    IF (Direction = ComDirection.ROB_TO_PLC)
    THEN  
      // calculate sequence payload length
      CalculateSequencePayloadMax := ( _parCfg.Com.TelegramLengthRobToPlc - _cyclicDataLength );
    END_IF
    

  SequenceFlag.SECONDARY_SEQUENCE :
  
    IF (Direction = ComDirection.PLC_TO_ROB)
    THEN  
      // calculate sequence payload length
      CalculateSequencePayloadMax := (( _parCfg.Com.TelegramLengthPlcToRob - _cyclicDataLength ) / 2);
    END_IF

    IF (Direction = ComDirection.ROB_TO_PLC)
    THEN  
      // calculate sequence payload length
      CalculateSequencePayloadMax := (( _parCfg.Com.TelegramLengthRobToPlc - _cyclicDataLength ) / 2);
    END_IF

    
END_CASE
                
END_METHOD

METHOD CalculateSequencePayloadStartAdr : UINT
VAR_IN_OUT
  /// Robot assignment of function
  AxesGroup : AxesGroup;
END_VAR
VAR_INPUT
  /// Communication direction
  Direction : ComDirection;
  /// Sequeunce
  Sequence : SequenceFlag;  
END_VAR

VAR
  /// Length of the cyclic header
 _cyclicDataLength      : UINT;
  /// Length of the sequnce payload
 _sequencePayloadLength : UINT;
END_VAR
                  // calculate cyclic header length
_cyclicDataLength := CalculateCyclicDataLength(AxesGroup := AxesGroup, Direction := Direction);

CASE (Sequence) 
OF

  SequenceFlag.PRIMARY_SEQUENCE   : 
  
    // return start address
    CalculateSequencePayloadStartAdr := _cyclicDataLength;

  SequenceFlag.SECONDARY_SEQUENCE :
  
    // calculate sequence payload max
   _sequencePayloadLength 
     := CalculateSequencePayloadMax( AxesGroup := AxesGroup, 
                                     Direction := Direction, 
                                     Sequence  := Sequence );
                                     
    // return start address
    CalculateSequencePayloadStartAdr := _cyclicDataLength + _sequencePayloadLength;
    
END_CASE
                
END_METHOD

METHOD PRIVATE CalculateTelegramLengthPlcToRob : UINT
VAR_IN_OUT
  /// Robot assignment of function
  AxesGroup : AxesGroup;
END_VAR
VAR
  /// length of the cyclic data block
 _cyclicDataLength : UINT;
END_VAR
                  _cyclicDataLength := CalculateCyclicDataLength(AxesGroup := AxesGroup, Direction := ComDirection.PLC_TO_ROB); 


IF ( _parCfg.Com.TwoSequences )
THEN
  CalculateTelegramLengthPlcToRob := _cyclicDataLength
                                    + SIZEOF(Telegram.PlcToRob.Sequence[  PRIMARY_SEQUENCE].Header)
                                    +       (Telegram.PlcToRob.Sequence[  PRIMARY_SEQUENCE].Header.PayloadLength)
                                    + SIZEOF(Telegram.PlcToRob.Sequence[SECONDARY_SEQUENCE].Header)
                                    +       (Telegram.PlcToRob.Sequence[SECONDARY_SEQUENCE].Header.PayloadLength)
                                    + SIZEOF(Telegram.PlcToRob.Footer);  
ELSE
  CalculateTelegramLengthPlcToRob := _cyclicDataLength
                                    + SIZEOF(Telegram.PlcToRob.Sequence[PRIMARY_SEQUENCE].Header)
                                    +       (Telegram.PlcToRob.Sequence[PRIMARY_SEQUENCE].Header.PayloadLength)
                                    + SIZEOF(Telegram.PlcToRob.Footer);
END_IF
                
END_METHOD

METHOD PROTECTED CheckParameterChanged : BOOL
VAR_IN_OUT
  /// Robot assignment of function
  AxesGroup    : AxesGroup; 
END_VAR

VAR
  /// internal index for loops
 _idx : DINT;
END_VAR
                  // Check initialization is already done ?
IF ( NOT Initialized )
THEN
  CheckParameterChanged := FALSE;
  RETURN;
END_IF

// compare memory 
CheckParameterChanged := ( SysDepMemCmp(pData1 := ADR(ParCfg), pData2 := ADR(_parCfg), DataLen := SIZEOF(ParCfg)) <> RobotLibraryConstants.OK );

FOR _idx := SyncTime.DURING_START_UP TO SyncTime.AFTER_START_UP
DO
  // Check Tool SyncMode changed ? 
  IF ( _parCfg.Plc.Parameter.SynchronizationModes.Tool[_idx] <> ParCfg.Plc.Parameter.SynchronizationModes.Tool[_idx] )
  THEN
    // Set info
    SetInfo( InfoID := RobotLibraryInfoIdEnum.INFO_CHANGE_TOOL_SYNC_MODE_TO_NEGATIVE_ONLY_AT_PLC_START_ALLOWED, Overwrite := TRUE);
     
    // Create log entry
    CreateLogMessagePara3( Timestamp   := SystemTime,
                           MessageType := MessageType.CMD,
                           Severity    := Severity.INFO,
                           MessageCode := 0,
                           MessageText := 'SyncMode.Tool[{1}] changed from {2} to {3}, but this is only allowed at PLC start',
                           Para1       := SYNC_TIME_TO_STRING(_idx),
                           Para2       := SYNC_MODE_TO_STRING( ParCfg.Plc.Parameter.SynchronizationModes.Tool[_idx]),
                           Para3       := SYNC_MODE_TO_STRING(_parCfg.Plc.Parameter.SynchronizationModes.Tool[_idx]));   
  END_IF
  
  
  // Check Frame SyncMode changed ? 
  IF ( _parCfg.Plc.Parameter.SynchronizationModes.Frame[_idx] <> ParCfg.Plc.Parameter.SynchronizationModes.Frame[_idx] )
  THEN
    // Set info
    SetInfo( InfoID := RobotLibraryInfoIdEnum.INFO_CHANGE_FRAME_SYNC_MODE_TO_NEGATIVE_ONLY_AT_PLC_START_ALLOWED, Overwrite :=  TRUE);
     
    // Create log entry
    CreateLogMessagePara3( Timestamp   := SystemTime,
                           MessageType := MessageType.CMD,
                           Severity    := Severity.INFO,
                           MessageCode := 0,
                           MessageText := 'SyncMode.Frame[{1}] changed from {2} to {3}, but this is only allowed at PLC start',
                           Para1       := SYNC_TIME_TO_STRING(_idx),
                           Para2       := SYNC_MODE_TO_STRING( ParCfg.Plc.Parameter.SynchronizationModes.Frame[_idx]),
                           Para3       := SYNC_MODE_TO_STRING(_parCfg.Plc.Parameter.SynchronizationModes.Frame[_idx]));   
  END_IF
  
  
  // Check Load SyncMode changed ? 
  IF ( _parCfg.Plc.Parameter.SynchronizationModes.Load[_idx] <> ParCfg.Plc.Parameter.SynchronizationModes.Load[_idx] )
  THEN
    // Set info
    SetInfo( InfoID := RobotLibraryInfoIdEnum.INFO_CHANGE_LOAD_SYNC_MODE_TO_NEGATIVE_ONLY_AT_PLC_START_ALLOWED, Overwrite := TRUE);
     
    // Create log entry
    CreateLogMessagePara3( Timestamp   := SystemTime,
                           MessageType := MessageType.CMD,
                           Severity    := Severity.INFO,
                           MessageCode := 0,
                           MessageText := 'SyncMode.Load[{1}] changed from {2} to {3}, but this is only allowed at PLC start',
                           Para1       := SYNC_TIME_TO_STRING(_idx),
                           Para2       := SYNC_MODE_TO_STRING( ParCfg.Plc.Parameter.SynchronizationModes.Load[_idx]),
                           Para3       := SYNC_MODE_TO_STRING(_parCfg.Plc.Parameter.SynchronizationModes.Load[_idx]));   
  END_IF
  
  
  // Check WorkAreas SyncMode changed ? 
  IF ( _parCfg.Plc.Parameter.SynchronizationModes.WorkAreas[_idx] <> ParCfg.Plc.Parameter.SynchronizationModes.WorkAreas[_idx] )
  THEN
    // Set info
    SetInfo( InfoID := RobotLibraryInfoIdEnum.INFO_CHANGE_WORK_AREA_SYNC_MODE_TO_NEGATIVE_ONLY_AT_PLC_START_ALLOWED, Overwrite := TRUE);
     
    // Create log entry
    CreateLogMessagePara3( Timestamp   := SystemTime,
                           MessageType := MessageType.CMD,
                           Severity    := Severity.INFO,
                           MessageCode := 0,
                           MessageText := 'SyncMode.WorkAreas[{1}] changed from {2} to {3}, but this is only allowed at PLC start',
                           Para1       := SYNC_TIME_TO_STRING(_idx),
                           Para2       := SYNC_MODE_TO_STRING( ParCfg.Plc.Parameter.SynchronizationModes.WorkAreas[_idx]),
                           Para3       := SYNC_MODE_TO_STRING(_parCfg.Plc.Parameter.SynchronizationModes.WorkAreas[_idx]));   
  END_IF

  // Check SWLimits SyncMode changed ? 
  IF ( _parCfg.Plc.Parameter.SynchronizationModes.SWLimits[_idx] <> ParCfg.Plc.Parameter.SynchronizationModes.SWLimits[_idx] )
  THEN
    // Set info
    SetInfo( InfoID := RobotLibraryInfoIdEnum.INFO_CHANGE_SWLIMITS_SYNC_MODE_TO_NEGATIVE_ONLY_AT_PLC_START_ALLOWED, Overwrite := TRUE);
     
    // Create log entry
    CreateLogMessagePara3( Timestamp   := SystemTime,
                           MessageType := MessageType.CMD,
                           Severity    := Severity.INFO,
                           MessageCode := 0,
                           MessageText := 'SyncMode.SWLimits[{1}] changed from {2} to {3}, but this is only allowed at PLC start',
                           Para1       := SYNC_TIME_TO_STRING(_idx),
                           Para2       := SYNC_MODE_TO_STRING( ParCfg.Plc.Parameter.SynchronizationModes.SWLimits[_idx]),
                           Para3       := SYNC_MODE_TO_STRING(_parCfg.Plc.Parameter.SynchronizationModes.SWLimits[_idx]));   
  END_IF
  
 
  // Check DefaultDynamics SyncMode changed ? 
  IF ( _parCfg.Plc.Parameter.SynchronizationModes.DefaultDynamics[_idx] <> ParCfg.Plc.Parameter.SynchronizationModes.DefaultDynamics[_idx] )
  THEN
    // Set info
    SetInfo( InfoID := RobotLibraryInfoIdEnum.INFO_CHANGE_DEFAULT_DYNAMICS_SYNC_MODE_TO_NEGATIVE_ONLY_AT_PLC_START_ALLOWED, Overwrite := TRUE);
     
    // Create log entry
    CreateLogMessagePara3( Timestamp   := SystemTime,
                           MessageType := MessageType.CMD,
                           Severity    := Severity.INFO,
                           MessageCode := 0,
                           MessageText := 'SyncMode.DefaultDynamics[{1}] changed from {2} to {3}, but this is only allowed at PLC start',
                           Para1       := SYNC_TIME_TO_STRING(_idx),
                           Para2       := SYNC_MODE_TO_STRING( ParCfg.Plc.Parameter.SynchronizationModes.DefaultDynamics[_idx]),
                           Para3       := SYNC_MODE_TO_STRING(_parCfg.Plc.Parameter.SynchronizationModes.DefaultDynamics[_idx]));   
  END_IF
  
  
  // Check ReferenceDynamics SyncMode changed ?
  IF ( _parCfg.Plc.Parameter.SynchronizationModes.ReferenceDynamics[_idx] <> ParCfg.Plc.Parameter.SynchronizationModes.ReferenceDynamics[_idx] )
  THEN
    // Set info
    SetInfo(InfoID := RobotLibraryInfoIdEnum.INFO_CHANGE_REFERENCE_DYNAMICS_SYNC_MODE_TO_NEGATIVE_ONLY_AT_PLC_START_ALLOWED, Overwrite := TRUE );
     
    // Create log entry
    CreateLogMessagePara3( Timestamp   := SystemTime,
                           MessageType := MessageType.CMD,
                           Severity    := Severity.INFO,
                           MessageCode := 0,
                           MessageText := 'SyncMode.ReferenceDynamics[{1}] changed from {2} to {3}, but this is only allowed at PLC start',
                           Para1       := SYNC_TIME_TO_STRING(_idx),
                           Para2       := SYNC_MODE_TO_STRING( ParCfg.Plc.Parameter.SynchronizationModes.ReferenceDynamics[_idx]),
                           Para3       := SYNC_MODE_TO_STRING(_parCfg.Plc.Parameter.SynchronizationModes.ReferenceDynamics[_idx]));   
  END_IF

END_FOR


// Check Plc.OptionalCyclic changed ? 
IF ( PlcOptionalCyclicToUint(_parCfg.Plc.OptionalCyclic) <> PlcOptionalCyclicToUint(ParCfg.Plc.OptionalCyclic ))
THEN
  // Set error
  SetError( ErrorID := RobotLibraryErrorIdEnum.ERR_TELEGRAM_NUMBER_CHANGED_AFTER_INIT, Overwrite := TRUE );
   
  // Create log entry
  CreateLogMessagePara2( Timestamp   := SystemTime,
                         MessageType := MessageType.CMD,
                         Severity    := Severity.ERROR,
                         MessageCode := 0,
                         MessageText := 'ParCfg.Plc.OptionalCyclic changed after initialization from {1} to {2} -> Reinitialize by disabling and enabling the RobotTask',
                         Para1       := WORD_TO_STRING_BIN(PlcOptionalCyclicToUint(_parCfg.Plc.OptionalCyclic)),
                         Para2       := WORD_TO_STRING_BIN(PlcOptionalCyclicToUint( ParCfg.Plc.OptionalCyclic)));   
END_IF


// Check Rob.OptionalCyclic changed ? 
IF ( RobOptionalCyclicToUint(_parCfg.Rob.OptionalCyclic) <> RobOptionalCyclicToUint(ParCfg.Rob.OptionalCyclic ))
THEN
  // Set error
  SetError( ErrorID := RobotLibraryErrorIdEnum.ERR_TELEGRAM_NUMBER_CHANGED_AFTER_INIT, Overwrite := TRUE );
   
  // Create log entry
  CreateLogMessagePara2( Timestamp   := SystemTime,
                         MessageType := MessageType.CMD,
                         Severity    := Severity.ERROR,
                         MessageCode := 0,
                         MessageText := 'ParCfg.Rob.OptionalCyclic changed after initialization from {1} to {2} -> Reinitialize by disabling and enabling the RobotTask',
                         Para1       := WORD_TO_STRING_BIN(RobOptionalCyclicToUint(_parCfg.Rob.OptionalCyclic)),
                         Para2       := WORD_TO_STRING_BIN(RobOptionalCyclicToUint( ParCfg.Rob.OptionalCyclic)));   
END_IF

                
END_METHOD

METHOD PROTECTED CheckParameterValid : BOOL
VAR_IN_OUT
  /// Robot assignment of function
  AxesGroup : AxesGroup; 
END_VAR
                  // init return value
CheckParameterValid := TRUE;


// Check ParCfg.Com.TelegramLengthPlcToRob
IF ( ParCfg.Com.TelegramLengthPlcToRob < 128 )
THEN
  // Set Warning
  SetWarning( WarningID := RobotLibraryWarningIdEnum.WARN_ACYCLIC_RANGE_PLC_TO_ROB_VERY_SMALL, Overwrite := TRUE );
END_IF

// Check ParCfg.Com.TelegramLengthRobToPlc
IF ( ParCfg.Com.TelegramLengthRobToPlc < 128 )
THEN
  // Set Warning
  SetWarning( WarningID := RobotLibraryWarningIdEnum.WARN_ACYCLIC_RANGE_ROB_TO_PLC_VERY_SMALL, Overwrite := TRUE );
END_IF



// Region ParCfg.Com {{{

// Check LifeSignTimeout
IF ( ParCfg.Com.LifeSignTimeOut < T#10MS )
THEN
  // set to valid min value
  ParCfg.Com.LifeSignTimeOut := T#10MS;
 
  // Set info
  SetInfo( InfoID := RobotLibraryInfoIdEnum.INFO_LIFESIGN_TIMEOUT_TO_SMALL_AND_SET_TO_10MS, Overwrite := TRUE);
   
  // Create log entry
  CreateLogMessagePara1 ( Timestamp   := SystemTime,
                          MessageType := MessageType.CMD,
                          Severity    := Severity.INFO,
                          MessageCode := 0,
                          MessageText := 'LifeSignTimeout to small and set from {1}ms to 10ms',
                          Para1       := TIME_TO_STRING(ParCfg.Com.LifeSignTimeOut));                          
END_IF


// Check ParCfg.Com.TelegramLengthPlcToRob
IF (( ParCfg.Com.TelegramLengthPlcToRob < 64                  ) OR
    ( ParCfg.Com.TelegramLengthPlcToRob > ROBOT_OUT_DATA_SIZE ))
THEN
  // parameter(s) not valid
  CheckParameterValid := FALSE;

  // Set error
  SetError( ErrorID := RobotLibraryErrorIdEnum.ERR_TELEGRAM_LENGTH_MISMATCH_0x80A3, Overwrite := TRUE );
   
  // Create log entry
  CreateLogMessagePara1 ( Timestamp   := SystemTime,
                          MessageType := MessageType.CMD,
                          Severity    := Severity.INFO,
                          MessageCode := 0,
                          MessageText :=               'ParCfg.Com.TelegramLengthPlcToRob {1} invalid',
                          Para1       := UINT_TO_STRING(ParCfg.Com.TelegramLengthPlcToRob));
  // no further validation                          
  RETURN;                          
END_IF

// Check ParCfg.Com.TelegramLengthRobToPlc
IF (( ParCfg.Com.TelegramLengthRobToPlc < 64                 ) OR
    ( ParCfg.Com.TelegramLengthRobToPlc > ROBOT_IN_DATA_SIZE ))
THEN
  // parameter(s) not valid
  CheckParameterValid := FALSE;

  // Set error
  SetError( ErrorID := RobotLibraryErrorIdEnum.ERR_TELEGRAM_LENGTH_MISMATCH_0x80A3, Overwrite := TRUE );
   
  // Create log entry
  CreateLogMessagePara1 ( Timestamp   := SystemTime,
                          MessageType := MessageType.CMD,
                          Severity    := Severity.INFO,
                          MessageCode := 0,
                          MessageText :=               'ParCfg.Com.TelegramLengthRobToPlc {1} invalid',
                          Para1       := UINT_TO_STRING(ParCfg.Com.TelegramLengthRobToPlc));
  // no further validation                          
  RETURN;                          
END_IF
// EndRegion }}}

// Region ParCfg.Rob.OptionalCyclic {{{

// Check configuration if optional cyclic CartesianPosition valid ?
IF ( ParCfg.Rob.OptionalCyclic.UseCartesianPosition AND ParCfg.Rob.OptionalCyclic.UseCartesianPositionExt )
THEN
  // set to valid configuration
  ParCfg.Rob.OptionalCyclic.UseCartesianPosition    := TRUE;
  ParCfg.Rob.OptionalCyclic.UseCartesianPositionExt := FALSE;
 
  // Set info
  SetInfo( InfoID := RobotLibraryInfoIdEnum.INFO_RECV_EXT_CART_POS_NOT_USABLE_WITH_RECV_CART_POS, Overwrite := TRUE);
   
  // Create log entry
  CreateLogMessage( Timestamp   := SystemTime,
                    MessageType := MessageType.CMD,
                    Severity    := Severity.INFO,
                    MessageCode := 0,
                    MessageText := 'UseCartesianPosition and UseCartesianPositionExt cannot be configured together -> UseCartesianPosition is automatically activated');
END_IF


// Check configuration if optional cyclic JointPosition valid ?
IF ( ParCfg.Rob.OptionalCyclic.UseJointPosition AND ParCfg.Rob.OptionalCyclic.UseJointPositionExt ) AND FALSE  {warning 'ToDo: Yaskawa need this combination for debugging via JointPosExt '}
THEN
  // set to valid configuration
  ParCfg.Rob.OptionalCyclic.UseJointPosition    := TRUE;
  ParCfg.Rob.OptionalCyclic.UseJointPositionExt := FALSE;
 
  // Set info
  SetInfo( InfoID := RobotLibraryInfoIdEnum.INFO_RECV_EXT_JOINT_POS_NOT_USABLE_WITH_RECV_JOINT_POS, Overwrite := TRUE);
   
  // Create log entry
  CreateLogMessage( Timestamp   := SystemTime,
                    MessageType := MessageType.CMD,
                    Severity    := Severity.INFO,
                    MessageCode := 0,
                    MessageText := 'UseJointPosition and UseJointPositionExt cannot be configured together -> UseJointPosition is automatically activated');
END_IF
// EndRegion }}}

// Region ParCfg.Parameter.SynchronizationModes {{{

// Check ToolData synchronisation mode during startup
IF (( ParCfg.Plc.Parameter.SynchronizationModes.Tool[SyncTime.DURING_START_UP] <  SyncMode.NO_SYNCHRONIZATION ) OR
    ( ParCfg.Plc.Parameter.SynchronizationModes.Tool[SyncTime.DURING_START_UP] >= SyncMode.AUTOMATIC          )) // Automatic is not allowed during startup
THEN
  // parameter(s) not valid
  CheckParameterValid := FALSE;
 
  // Set error
  SetError  ( ErrorID   := RobotLibraryErrorIdEnum.ERR_SYNC_MODE_INVALID             , Overwrite := TRUE ); // own defined error - not in specification
  // Set warning
  SetWarning( WarningID := RobotLibraryWarningIdEnum.WARN_TOOL_DATA_SYNC_MODE_INVALID, Overwrite := TRUE );
   
  // Create log entry
  CreateLogMessagePara1 ( Timestamp   := SystemTime,
                          MessageType := MessageType.CMD,
                          Severity    := Severity.INFO,
                          MessageCode := 0,
                          MessageText :=                    'ParCfg.Plc.Parameter.SynchronizationModes.Tool[SyncTime.DURING_START_UP] invalid SyncMode {1}',
                          Para1       := SYNC_MODE_TO_STRING(ParCfg.Plc.Parameter.SynchronizationModes.Tool[SyncTime.DURING_START_UP]));
  // no further validation                          
  RETURN;                                                    
END_IF

// Check ToolData synchronisation mode after startup
IF (( ParCfg.Plc.Parameter.SynchronizationModes.Tool[SyncTime.AFTER_START_UP] < SyncMode.NO_SYNCHRONIZATION ) OR
    ( ParCfg.Plc.Parameter.SynchronizationModes.Tool[SyncTime.AFTER_START_UP] > SyncMode.AUTOMATIC          ))
THEN
  // parameter(s) not valid
  CheckParameterValid := FALSE;
 
  // Set error
  SetError  ( ErrorID   := RobotLibraryErrorIdEnum.ERR_SYNC_MODE_INVALID             , Overwrite := TRUE); // own defined error - not in specification
  // Set warning
  SetWarning( WarningID := RobotLibraryWarningIdEnum.WARN_TOOL_DATA_SYNC_MODE_INVALID, Overwrite := TRUE);
   
  // Create log entry
  CreateLogMessagePara1 ( Timestamp   := SystemTime,
                          MessageType := MessageType.CMD,
                          Severity    := Severity.INFO,
                          MessageCode := 0,
                          MessageText :=                    'ParCfg.Plc.Parameter.SynchronizationModes.Tool[SyncTime.AFTER_START_UP] invalid SyncMode {1}',
                          Para1       := SYNC_MODE_TO_STRING(ParCfg.Plc.Parameter.SynchronizationModes.Tool[SyncTime.AFTER_START_UP]));
  // no further validation                          
  RETURN;                                                    
END_IF


// Check FrameData synchronisation mode during startup
IF (( ParCfg.Plc.Parameter.SynchronizationModes.Frame[SyncTime.DURING_START_UP] <  SyncMode.NO_SYNCHRONIZATION ) OR
    ( ParCfg.Plc.Parameter.SynchronizationModes.Frame[SyncTime.DURING_START_UP] >= SyncMode.AUTOMATIC          )) // Automatic is not allowed during startup
THEN
  // parameter(s) not valid
  CheckParameterValid := FALSE;
 
  // Set error
  SetError  ( ErrorID   := RobotLibraryErrorIdEnum.ERR_SYNC_MODE_INVALID              , Overwrite := TRUE);// own defined error - not in specification
  // Set warning
  SetWarning( WarningID := RobotLibraryWarningIdEnum.WARN_FRAME_DATA_SYNC_MODE_INVALID, Overwrite := FALSE);
   
  // Create log entry
  CreateLogMessagePara1 ( Timestamp   := SystemTime,
                          MessageType := MessageType.CMD,
                          Severity    := Severity.INFO,
                          MessageCode := 0,
                          MessageText :=                    'ParCfg.Plc.Parameter.SynchronizationModes.Frame[SyncTime.DURING_START_UP] invalid SyncMode {1}',
                          Para1       := SYNC_MODE_TO_STRING(ParCfg.Plc.Parameter.SynchronizationModes.Frame[SyncTime.DURING_START_UP]));
  // no further validation                          
  RETURN;                                                   
END_IF


// Check FrameData synchronisation mode after startup
IF (( ParCfg.Plc.Parameter.SynchronizationModes.Frame[SyncTime.AFTER_START_UP] < SyncMode.NO_SYNCHRONIZATION ) OR
    ( ParCfg.Plc.Parameter.SynchronizationModes.Frame[SyncTime.AFTER_START_UP] > SyncMode.AUTOMATIC          ))
THEN
  // parameter(s) not valid
  CheckParameterValid := FALSE;
 
  // Set error
  SetError  ( ErrorID   := RobotLibraryErrorIdEnum.ERR_SYNC_MODE_INVALID              , Overwrite := TRUE);// own defined error - not in specification
  // Set warning
  SetWarning( WarningID := RobotLibraryWarningIdEnum.WARN_FRAME_DATA_SYNC_MODE_INVALID, Overwrite := TRUE);
   
  // Create log entry
  CreateLogMessagePara1 ( Timestamp   := SystemTime,
                          MessageType := MessageType.CMD,
                          Severity    := Severity.INFO,
                          MessageCode := 0,
                          MessageText :=                    'ParCfg.Plc.Parameter.SynchronizationModes.Frame[SyncTime.AFTER_START_UP] invalid SyncMode {1}',
                          Para1       := SYNC_MODE_TO_STRING(ParCfg.Plc.Parameter.SynchronizationModes.Frame[SyncTime.AFTER_START_UP]));
  // no further validation                          
  RETURN;                                                    
END_IF


// Check LoadData synchronisation mode during startup
IF (( ParCfg.Plc.Parameter.SynchronizationModes.Load[SyncTime.DURING_START_UP] <  SyncMode.NO_SYNCHRONIZATION ) OR
    ( ParCfg.Plc.Parameter.SynchronizationModes.Load[SyncTime.DURING_START_UP] >= SyncMode.AUTOMATIC          )) // Automatic is not allowed during startup
THEN
  // parameter(s) not valid
  CheckParameterValid := FALSE;
 
  // Set error
  SetError   ( ErrorID   := RobotLibraryErrorIdEnum.ERR_SYNC_MODE_INVALID             , Overwrite := TRUE);// own defined error - not in specification
  // Set warning
  SetWarning ( WarningID := RobotLibraryWarningIdEnum.WARN_LOAD_DATA_SYNC_MODE_INVALID, Overwrite := TRUE);
   
  // Create log entry
  CreateLogMessagePara1 ( Timestamp   := SystemTime,
                          MessageType := MessageType.CMD,
                          Severity    := Severity.INFO,
                          MessageCode := 0,
                          MessageText :=                    'ParCfg.Plc.Parameter.SynchronizationModes.Load[SyncTime.DURING_START_UP] invalid SyncMode {1}',
                          Para1       := SYNC_MODE_TO_STRING(ParCfg.Plc.Parameter.SynchronizationModes.Load[SyncTime.DURING_START_UP]));
  // no further validation                          
  RETURN;                          
END_IF


// Check LoadData synchronisation mode after startup
IF (( ParCfg.Plc.Parameter.SynchronizationModes.Load[SyncTime.AFTER_START_UP] < SyncMode.NO_SYNCHRONIZATION ) OR
    ( ParCfg.Plc.Parameter.SynchronizationModes.Load[SyncTime.AFTER_START_UP] > SyncMode.AUTOMATIC          ))
THEN
  // parameter(s) not valid
  CheckParameterValid := FALSE;
 
  // Set error
  SetError  ( ErrorID   := RobotLibraryErrorIdEnum.ERR_SYNC_MODE_INVALID,              Overwrite := TRUE);// own defined error - not in specification
  // Set warning
  SetWarning( WarningID := RobotLibraryWarningIdEnum.WARN_LOAD_DATA_SYNC_MODE_INVALID, Overwrite := TRUE);
   
  // Create log entry
  CreateLogMessagePara1 ( Timestamp   := SystemTime,
                          MessageType := MessageType.CMD,
                          Severity    := Severity.INFO,
                          MessageCode := 0,
                          MessageText :=                    'ParCfg.Plc.Parameter.SynchronizationModes.Load[SyncTime.AFTER_START_UP] invalid SyncMode {1}',
                          Para1       := SYNC_MODE_TO_STRING(ParCfg.Plc.Parameter.SynchronizationModes.Load[SyncTime.AFTER_START_UP]));
  // no further validation                          
  RETURN;                          
END_IF


// Check WorkAreas synchronisation mode during startup
IF (( ParCfg.Plc.Parameter.SynchronizationModes.WorkAreas[SyncTime.DURING_START_UP] <  SyncMode.NO_SYNCHRONIZATION ) OR
    ( ParCfg.Plc.Parameter.SynchronizationModes.WorkAreas[SyncTime.DURING_START_UP] >= SyncMode.AUTOMATIC          )) // Automatic is not allowed during startup
THEN
  // parameter(s) not valid
  CheckParameterValid := FALSE;
 
  // Set error
  SetError  ( ErrorID   := RobotLibraryErrorIdEnum.ERR_SYNC_MODE_INVALID,              Overwrite := TRUE);// own defined error - not in specification
  // Set warning
  SetWarning( WarningID := RobotLibraryWarningIdEnum.WARN_WORK_AREA_SYNC_MODE_INVALID, Overwrite := TRUE);
   
  // Create log entry
  CreateLogMessagePara1 ( Timestamp   := SystemTime,
                          MessageType := MessageType.CMD,
                          Severity    := Severity.INFO,
                          MessageCode := 0,
                          MessageText :=                    'ParCfg.Plc.Parameter.SynchronizationModes.WorkAreas[SyncTime.DURING_START_UP] invalid SyncMode {1}',
                          Para1       := SYNC_MODE_TO_STRING(ParCfg.Plc.Parameter.SynchronizationModes.WorkAreas[SyncTime.DURING_START_UP]));
  // no further validation                          
  RETURN;                          
END_IF


// Check WorkAreas synchronisation mode after startup
IF (( ParCfg.Plc.Parameter.SynchronizationModes.WorkAreas[SyncTime.AFTER_START_UP] < SyncMode.NO_SYNCHRONIZATION ) OR
    ( ParCfg.Plc.Parameter.SynchronizationModes.WorkAreas[SyncTime.AFTER_START_UP] > SyncMode.AUTOMATIC          ))
THEN
  // parameter(s) not valid
  CheckParameterValid := FALSE;
 
  // Set error
  SetError  ( ErrorID   := RobotLibraryErrorIdEnum.ERR_SYNC_MODE_INVALID,              Overwrite := TRUE);// own defined error - not in specification
  // Set warning
  SetWarning( WarningID := RobotLibraryWarningIdEnum.WARN_WORK_AREA_SYNC_MODE_INVALID, Overwrite := TRUE);
   
  // Create log entry
  CreateLogMessagePara1 ( Timestamp   := SystemTime,
                          MessageType := MessageType.CMD,
                          Severity    := Severity.INFO,
                          MessageCode := 0,
                          MessageText :=                    'ParCfg.Plc.Parameter.SynchronizationModes.WorkAreas[SyncTime.AFTER_START_UP] invalid SyncMode {1}',
                          Para1       := SYNC_MODE_TO_STRING(ParCfg.Plc.Parameter.SynchronizationModes.WorkAreas[SyncTime.AFTER_START_UP]));
  // no further validation                          
  RETURN;                          
END_IF


// Check SWLimits synchronisation mode during startup
IF (( ParCfg.Plc.Parameter.SynchronizationModes.SWLimits[SyncTime.DURING_START_UP] <  SyncMode.NO_SYNCHRONIZATION ) OR
    ( ParCfg.Plc.Parameter.SynchronizationModes.SWLimits[SyncTime.DURING_START_UP] >= SyncMode.AUTOMATIC          )) // Automatic is not allowed during startup
THEN
  // parameter(s) not valid
  CheckParameterValid := FALSE;
 
  // Set error
  SetError  ( ErrorID   := RobotLibraryErrorIdEnum.ERR_SYNC_MODE_INVALID,              Overwrite := TRUE);// own defined error - not in specification
  // Set warning
  SetWarning( WarningID := RobotLibraryWarningIdEnum.WARN_SW_LIMITS_SYNC_MODE_INVALID, Overwrite := TRUE);
   
  // Create log entry
  CreateLogMessagePara1 ( Timestamp   := SystemTime,
                          MessageType := MessageType.CMD,
                          Severity    := Severity.INFO,
                          MessageCode := 0,
                          MessageText :=                    'ParCfg.Plc.Parameter.SynchronizationModes.SWLimits[SyncTime.DURING_START_UP] invalid SyncMode {1}',
                          Para1       := SYNC_MODE_TO_STRING(ParCfg.Plc.Parameter.SynchronizationModes.SWLimits[SyncTime.DURING_START_UP]));
  // no further validation                          
  RETURN;                          
END_IF


// Check SWLimits synchronisation mode after startup
IF (( ParCfg.Plc.Parameter.SynchronizationModes.SWLimits[SyncTime.AFTER_START_UP] < SyncMode.NO_SYNCHRONIZATION ) OR
    ( ParCfg.Plc.Parameter.SynchronizationModes.SWLimits[SyncTime.AFTER_START_UP] > SyncMode.AUTOMATIC          ))
THEN
  // parameter(s) not valid
  CheckParameterValid := FALSE;
 
  // Set error
  SetError  ( ErrorID   := RobotLibraryErrorIdEnum.ERR_SYNC_MODE_INVALID,              Overwrite := TRUE);// own defined error - not in specification
  // Set warning
  SetWarning( WarningID := RobotLibraryWarningIdEnum.WARN_SW_LIMITS_SYNC_MODE_INVALID, Overwrite := TRUE);
   
  // Create log entry
  CreateLogMessagePara1 ( Timestamp   := SystemTime,
                          MessageType := MessageType.CMD,
                          Severity    := Severity.INFO,
                          MessageCode := 0,
                          MessageText :=                    'ParCfg.Plc.Parameter.SynchronizationModes.SWLimits[SyncTime.AFTER_START_UP] invalid SyncMode {1}',
                          Para1       := SYNC_MODE_TO_STRING(ParCfg.Plc.Parameter.SynchronizationModes.SWLimits[SyncTime.AFTER_START_UP]));
  // no further validation                          
  RETURN;                          
END_IF


// Check DefaultDynamics synchronisation mode during startup
IF (( ParCfg.Plc.Parameter.SynchronizationModes.DefaultDynamics[SyncTime.DURING_START_UP] <  SyncMode.NO_SYNCHRONIZATION ) OR
    ( ParCfg.Plc.Parameter.SynchronizationModes.DefaultDynamics[SyncTime.DURING_START_UP] >= SyncMode.AUTOMATIC          )) // Automatic is not allowed during startup
THEN
  // parameter(s) not valid
  CheckParameterValid := FALSE;
 
  // Set error
  SetError  ( ErrorID   := RobotLibraryErrorIdEnum.ERR_SYNC_MODE_INVALID,                     Overwrite := TRUE);// own defined error - not in specification
  // Set warning
  SetWarning( WarningID := RobotLibraryWarningIdEnum.WARN_DEFAULT_DYNAMICS_SYNC_MODE_INVALID, Overwrite := TRUE);
   
  // Create log entry
  CreateLogMessagePara1 ( Timestamp   := SystemTime,
                          MessageType := MessageType.CMD,
                          Severity    := Severity.INFO,
                          MessageCode := 0,
                          MessageText :=                    'ParCfg.Plc.Parameter.SynchronizationModes.DefaultDynamics[SyncTime.DURING_START_UP] invalid SyncMode {1}',
                          Para1       := SYNC_MODE_TO_STRING(ParCfg.Plc.Parameter.SynchronizationModes.DefaultDynamics[SyncTime.DURING_START_UP]));
  // no further validation                          
  RETURN;                          
END_IF


// Check DefaultDynamics synchronisation mode after startup
IF (( ParCfg.Plc.Parameter.SynchronizationModes.DefaultDynamics[SyncTime.AFTER_START_UP] < SyncMode.NO_SYNCHRONIZATION ) OR
    ( ParCfg.Plc.Parameter.SynchronizationModes.DefaultDynamics[SyncTime.AFTER_START_UP] > SyncMode.AUTOMATIC          ))
THEN
  // parameter(s) not valid
  CheckParameterValid := FALSE;
 
  // Set error
  SetError  ( ErrorID   := RobotLibraryErrorIdEnum.ERR_SYNC_MODE_INVALID,                     Overwrite := TRUE);// own defined error - not in specification
  // Set warning
  SetWarning( WarningID := RobotLibraryWarningIdEnum.WARN_DEFAULT_DYNAMICS_SYNC_MODE_INVALID, Overwrite := TRUE);
   
  // Create log entry
  CreateLogMessagePara1 ( Timestamp   := SystemTime,
                          MessageType := MessageType.CMD,
                          Severity    := Severity.INFO,
                          MessageCode := 0,
                          MessageText :=                    'ParCfg.Plc.Parameter.SynchronizationModes.DefaultDynamics[SyncTime.AFTER_START_UP] invalid SyncMode {1}',
                          Para1       := SYNC_MODE_TO_STRING(ParCfg.Plc.Parameter.SynchronizationModes.DefaultDynamics[SyncTime.AFTER_START_UP]));
  // no further validation                          
  RETURN;                          
END_IF


// Check ReferenceDynamics synchronisation mode during startup
IF (( ParCfg.Plc.Parameter.SynchronizationModes.ReferenceDynamics[SyncTime.DURING_START_UP] <  SyncMode.NO_SYNCHRONIZATION ) OR
    ( ParCfg.Plc.Parameter.SynchronizationModes.ReferenceDynamics[SyncTime.DURING_START_UP] >= SyncMode.AUTOMATIC          )) // Automatic is not allowed during startup
THEN
  // parameter(s) not valid
  CheckParameterValid := FALSE;
 
  // Set error
  SetError  ( ErrorID   := RobotLibraryErrorIdEnum.ERR_SYNC_MODE_INVALID,                       Overwrite := TRUE);// own defined error - not in specification
  // Set warning
  SetWarning( WarningID := RobotLibraryWarningIdEnum.WARN_REFERENCE_DYNAMICS_SYNC_MODE_INVALID, Overwrite := TRUE);
   
  // Create log entry
  CreateLogMessagePara1 ( Timestamp   := SystemTime,
                          MessageType := MessageType.CMD,
                          Severity    := Severity.INFO,
                          MessageCode := 0,
                          MessageText :=                    'ParCfg.Plc.Parameter.SynchronizationModes.ReferenceDynamics[SyncTime.DURING_START_UP] invalid SyncMode {1}',
                          Para1       := SYNC_MODE_TO_STRING(ParCfg.Plc.Parameter.SynchronizationModes.ReferenceDynamics[SyncTime.DURING_START_UP]));
  // no further validation                          
  RETURN;                          
END_IF


// Check ReferenceDynamics synchronisation mode after startup
IF (( ParCfg.Plc.Parameter.SynchronizationModes.ReferenceDynamics[SyncTime.AFTER_START_UP] < SyncMode.NO_SYNCHRONIZATION ) OR
    ( ParCfg.Plc.Parameter.SynchronizationModes.ReferenceDynamics[SyncTime.AFTER_START_UP] > SyncMode.AUTOMATIC          ))
THEN
  // parameter(s) not valid
  CheckParameterValid := FALSE;
 
  // Set error
  SetError  ( ErrorID   := RobotLibraryErrorIdEnum.ERR_SYNC_MODE_INVALID,                       Overwrite := TRUE);// own defined error - not in specification
  // Set warning
  SetWarning( WarningID := RobotLibraryWarningIdEnum.WARN_REFERENCE_DYNAMICS_SYNC_MODE_INVALID, Overwrite := TRUE);
   
  // Create log entry
  CreateLogMessagePara1 ( Timestamp   := SystemTime,
                          MessageType := MessageType.CMD,
                          Severity    := Severity.INFO,
                          MessageCode := 0,
                          MessageText :=                    'ParCfg.Plc.Parameter.SynchronizationModes.ReferenceDynamics[SyncTime.AFTER_START_UP] invalid SyncMode {1}',
                          Para1       := SYNC_MODE_TO_STRING(ParCfg.Plc.Parameter.SynchronizationModes.ReferenceDynamics[SyncTime.AFTER_START_UP]));
  // no further validation                          
  RETURN;                          
END_IF
// EndRegion }}}

                
END_METHOD

METHOD PRIVATE CreateSendPayload : DINT
VAR_IN_OUT
  /// Robot assignment of function
  AxesGroup    : AxesGroup;
  /// Outputs of PLC for communication to RC
  RobotOutData : ARRAY[*] OF BYTE;
END_VAR
                  // ------------------------------------
// Fill SendData
// ------------------------------------
// Call SendData FB, update payload and size 
SendData( Payload := RobotOutData, PayLoadSize := ROBOT_OUT_DATA_SIZE);
// reset all variables and payload
SendData.Reset();

CreateSendPayloadHeader        ( AxesGroup := AxesGroup );
CreateSendPayloadCyclic        ( AxesGroup := AxesGroup );
CreateSendPayloadCyclicOptional( AxesGroup := AxesGroup );
CreateSendPayloadSequence      ( AxesGroup := AxesGroup );
CreateSendPayloadFooter        ( AxesGroup := AxesGroup );
CreateSendPayloadLogging       ( AxesGroup := AxesGroup );

// reset NewSEQ flag
AxesGroup.State.NewSEQ[0] := FALSE; {warning 'Test'}
                
END_METHOD

METHOD PRIVATE CreateSendPayloadCyclic : DINT
VAR_IN_OUT
  /// Robot assignment of function
  AxesGroup : AxesGroup;
END_VAR
                  SendData.AddByte(Telegram.PlcToRob.Cyclic.ToolNo);  
SendData.AddByte(Telegram.PlcToRob.Cyclic.FrameNo); 

                
END_METHOD

METHOD PRIVATE CreateSendPayloadCyclicOptional : DINT
VAR_IN_OUT
  /// Robot assignment of function
  AxesGroup : AxesGroup;
END_VAR

VAR 
  /// temporary byte
 _tmpByte   : BYTE;
END_VAR
                  // Telegram.PlcToRob.CyclicOptional.SubProgramData {{{
IF ( AxesGroup.CyclicOptional.PlcToRob.SubProgramData.Active )
THEN
  SendData.AddDataBlock( ADR(Telegram.PlcToRob.CyclicOptional.SubProgramData.Data), SIZEOF(Telegram.PlcToRob.CyclicOptional.SubProgramData.Data));  
END_IF
// }}}
    
// Telegram.PlcToRob.CyclicOptional.CartesianPos {{{
IF ( AxesGroup.CyclicOptional.PlcToRob.CartesianPosition.Active) 
THEN
  SendData.AddReal(Telegram.PlcToRob.CyclicOptional.CartesianPosition.X );
  SendData.AddReal(Telegram.PlcToRob.CyclicOptional.CartesianPosition.Y );
  SendData.AddReal(Telegram.PlcToRob.CyclicOptional.CartesianPosition.Z );
  SendData.AddReal(Telegram.PlcToRob.CyclicOptional.CartesianPosition.Rx);
  SendData.AddReal(Telegram.PlcToRob.CyclicOptional.CartesianPosition.Ry);
  SendData.AddReal(Telegram.PlcToRob.CyclicOptional.CartesianPosition.Rz);

 _tmpByte   := 0;
 _tmpByte.0 := Telegram.PlcToRob.CyclicOptional.CartesianPosition.Config.0;
 _tmpByte.1 := Telegram.PlcToRob.CyclicOptional.CartesianPosition.Config.1;
 _tmpByte.2 := Telegram.PlcToRob.CyclicOptional.CartesianPosition.Config.2;
 
  SendData.AddByte(_tmpByte);
          
  SendData.AddByte (Telegram.PlcToRob.CyclicOptional.CartesianPosition.Turns_J2_J1             );
  SendData.AddByte (Telegram.PlcToRob.CyclicOptional.CartesianPosition.Turns_J4_J3             );
  SendData.AddByte (Telegram.PlcToRob.CyclicOptional.CartesianPosition.Turns_J6_J5             );
  SendData.AddByte (Telegram.PlcToRob.CyclicOptional.CartesianPosition.Turns_E1                );
  SendData.AddReal (Telegram.PlcToRob.CyclicOptional.CartesianPosition.E1                      );
END_IF
// }}}

// Telegram.PlcToRob.CyclicOptional.JointPosition {{{
IF ( AxesGroup.CyclicOptional.PlcToRob.JointPosition.Active) 
THEN
  SendData.AddReal(Telegram.PlcToRob.CyclicOptional.JointPosition.J1);
  SendData.AddReal(Telegram.PlcToRob.CyclicOptional.JointPosition.J2);
  SendData.AddReal(Telegram.PlcToRob.CyclicOptional.JointPosition.J3);
  SendData.AddReal(Telegram.PlcToRob.CyclicOptional.JointPosition.J4);
  SendData.AddReal(Telegram.PlcToRob.CyclicOptional.JointPosition.J5);
  SendData.AddReal(Telegram.PlcToRob.CyclicOptional.JointPosition.J6);
  SendData.AddReal(Telegram.PlcToRob.CyclicOptional.JointPosition.E1);
END_IF
// }}}

// Telegram.PlcToRob.CyclicOptional.Force {{{
IF ( AxesGroup.CyclicOptional.PlcToRob.Force.Active) 
THEN
  SendData.AddReal(Telegram.PlcToRob.CyclicOptional.Force.X);
  SendData.AddReal(Telegram.PlcToRob.CyclicOptional.Force.Y);
  SendData.AddReal(Telegram.PlcToRob.CyclicOptional.Force.Z);
  SendData.AddReal(Telegram.PlcToRob.CyclicOptional.Force.Rx);
  SendData.AddReal(Telegram.PlcToRob.CyclicOptional.Force.Ry);
  SendData.AddReal(Telegram.PlcToRob.CyclicOptional.Force.Rz);
END_IF  
// }}}

// Telegram.PlcToRob.CyclicOptional.TwoSequences {{{
// }}}

// AxesGroup.OptionalCyclic.PlcToRob.CartesianPosExt {{{
IF ( AxesGroup.CyclicOptional.PlcToRob.CartesianPositionExt.Active) 
THEN
  SendData.AddReal(Telegram.PlcToRob.CyclicOptional.CartesianPositionExt.E2);
  SendData.AddReal(Telegram.PlcToRob.CyclicOptional.CartesianPositionExt.E3);
  SendData.AddReal(Telegram.PlcToRob.CyclicOptional.CartesianPositionExt.E4);
  SendData.AddReal(Telegram.PlcToRob.CyclicOptional.CartesianPositionExt.E5);
  SendData.AddReal(Telegram.PlcToRob.CyclicOptional.CartesianPositionExt.E6);
END_IF    
// }}}

// AxesGroup.OptionalCyclic.PlcToRob.JointPositionExt {{{
IF ( AxesGroup.CyclicOptional.PlcToRob.JointPositionExt.Active) 
THEN
  SendData.AddReal(Telegram.PlcToRob.CyclicOptional.JointPositionExt.E2);
  SendData.AddReal(Telegram.PlcToRob.CyclicOptional.JointPositionExt.E3);  
  SendData.AddReal(Telegram.PlcToRob.CyclicOptional.JointPositionExt.E4);
  SendData.AddReal(Telegram.PlcToRob.CyclicOptional.JointPositionExt.E5);
  SendData.AddReal(Telegram.PlcToRob.CyclicOptional.JointPositionExt.E6);        
END_IF  
// }}}
                    
// Telegram.PlcToRob.CyclicOptional..CartesianForceExt {{{
IF ( AxesGroup.CyclicOptional.PlcToRob.ForceExt.Active) 
THEN
  SendData.AddReal(Telegram.PlcToRob.CyclicOptional.ForceExt.E1);
  SendData.AddReal(Telegram.PlcToRob.CyclicOptional.ForceExt.E2);
  SendData.AddReal(Telegram.PlcToRob.CyclicOptional.ForceExt.E3);
  SendData.AddReal(Telegram.PlcToRob.CyclicOptional.ForceExt.E4);
  SendData.AddReal(Telegram.PlcToRob.CyclicOptional.ForceExt.E5);
  SendData.AddReal(Telegram.PlcToRob.CyclicOptional.ForceExt.E6);
END_IF                    
// }}}
                
END_METHOD

METHOD PRIVATE CreateSendPayloadFooter : DINT
VAR_IN_OUT
  /// Robot assignment of function
  AxesGroup : AxesGroup;
END_VAR
VAR
END_VAR
                  SendData.SetLifeSignFooter( LifeSign :=  AxesGroup.Cyclic.PlcToRob.LifeSign);

                
END_METHOD

METHOD PRIVATE CreateSendPayloadHeader : DINT
VAR_IN_OUT
  /// Robot assignment of function
  AxesGroup : AxesGroup;
END_VAR
                  SendData.AddByte(Telegram.PlcToRob.Header.SRCIVersion           );
SendData.AddByte(Telegram.PlcToRob.Header.FastStop_LifeSign     ); 
SendData.AddUint(Telegram.PlcToRob.Header.TelegramLengthPlcToRob);
SendData.AddUint(Telegram.PlcToRob.Header.TelegramLengthRobToPlc);
SendData.AddByte(Telegram.PlcToRob.Header.AxesGroupID_Control   );
SendData.AddByte(Telegram.PlcToRob.Header.Reserved              );
SendData.AddUint(Telegram.PlcToRob.Header.TelegramNumberPlcToRob);
SendData.AddUint(Telegram.PlcToRob.Header.TelegramNumberRobToPlc);
SendData.AddUint(Telegram.PlcToRob.Header.ClientDate            ); 
SendData.AddTime(Telegram.PlcToRob.Header.ClientTime            );  
                
END_METHOD

METHOD PRIVATE CreateSendPayloadLogging : DINT
VAR_IN_OUT
  /// Robot assignment of function
  AxesGroup                 : AxesGroup;
END_VAR
                  IF  ((( Telegram.PlcToRob.Sequence[0].Header.PayloadLength > 0 ) AND (AxesGroup.State.NewSEQ[0] )) OR
     (( Telegram.PlcToRob.Sequence[1].Header.PayloadLength > 0 ) AND (AxesGroup.State.NewSEQ[1] )))
THEN
  // Create log entry
  CreateLogMessagePara1 ( Timestamp   := SystemTime,
                          MessageType := MessageType.CMD,
                          Severity    := Severity.DEBUG,
                          MessageCode := 0,
                          MessageText := 'SendData: Bytes send in total: {1}',
                          Para1       :=  UDINT_TO_STRING(SendData.PayloadLen));
END_IF
                
END_METHOD

METHOD PRIVATE CreateSendPayloadSequence : DINT
VAR_IN_OUT
  /// Robot assignment of function
  AxesGroup                 : AxesGroup;
END_VAR

VAR 
  /// internal sequence index
 _seqIdx                    : DINT;
  /// internal fragment index
 _fragIdx                   : DINT;
END_VAR
                  FOR _seqIdx := 0 TO AxesGroup.State.SequenceCountSend
DO
  // Check 2nd sequence ? -> goto 2nd sequence payload address  
  IF ( _seqIdx = SECONDARY_SEQUENCE )
  THEN
    SendData.PayloadPtr := CalculateSequencePayloadStartAdr(AxesGroup := AxesGroup, 
                                                            Direction := ComDirection.PLC_TO_ROB,
                                                            Sequence  := SequenceFlag.SECONDARY_SEQUENCE);
  END_IF

  // Telegram.PlcToRob.Sequence[x].Header {{{
  SendData.AddUint(Telegram.PlcToRob.Sequence[_seqIdx].Header.SEQ_ACK);
  SendData.AddUint(Telegram.PlcToRob.Sequence[_seqIdx].Header.PayloadLength);
  // }}}

  // check limit reachted ?
  IF ( SendData.PayloadPtr + FOOTER_SIZE >= Telegram.PlcToRob.Header.TelegramLengthPlcToRob)
  THEN
    EXIT;
  END_IF
  
  // PlcToRob.Sequence[x].Fragment[x] {{{
  FOR _fragIdx := 0 TO AxesGroup.State.FragmentCountSend[_seqIdx]  
  DO

    IF (Telegram.PlcToRob.Sequence[_seqIdx].Fragment[_fragIdx].Header.PayloadLength > 0)
    THEN  
      // PlcToRob.Sequence[x].Fragment[x].Header {{{        
      SendData.AddUint(Telegram.PlcToRob.Sequence[_seqIdx].Fragment[_fragIdx].Header.CmdID);
      SendData.AddByte(Telegram.PlcToRob.Sequence[_seqIdx].Fragment[_fragIdx].Header.Reserve);
      SendData.AddByte(Telegram.PlcToRob.Sequence[_seqIdx].Fragment[_fragIdx].Header.FragmentAction);
      SendData.AddUint(Telegram.PlcToRob.Sequence[_seqIdx].Fragment[_fragIdx].Header.PayloadPointer);
      SendData.AddUint(Telegram.PlcToRob.Sequence[_seqIdx].Fragment[_fragIdx].Header.PayloadLength);
      // }}}
      
      // PlcToRob.Sequence[x].Fragment[x].Command {{{
      
      // Hint: the command header is part of the fragment payload  
      IF (Telegram.PlcToRob.Sequence[_seqIdx].Fragment[_fragIdx].Header.PayloadLength > 0)
      THEN
        SendData.AddDataBlock( pValue :=  ADR(Telegram.PlcToRob.Sequence[_seqIdx].Fragment[_fragIdx].Command.Payload           ) + Telegram.PlcToRob.Sequence[_seqIdx].Fragment[_fragIdx].Header.PayloadPointer,
                                 Size :=     (Telegram.PlcToRob.Sequence[_seqIdx].Fragment[_fragIdx].Header.PayloadLength      ));

      END_IF
      
      
      IF (SendData.PayloadLen = 232)
      THEN
        SendData.PayloadLen := SendData.PayloadLen;
			END_IF
      
    END_IF
    // }}}
  END_FOR
  // }}}
END_FOR  
                
END_METHOD

METHOD FB_init : BOOL
VAR_INPUT
  bInitRetains : BOOL; // if TRUE, the retain variables are initialized (warm start / cold start)
  bInCopyCode : BOOL;  // if TRUE, the instance afterwards gets moved into the copy code (online change)
END_VAR
                  MyType := 'MC_RobotTaskFB';

// Create log entry
CreateLogMessage ( Timestamp   := SystemTime,
                   MessageType := MessageType.CMD,
                   Severity    := Severity.DEBUG,
                   MessageCode := 0,
                   MessageText := 'PLC started / restarted');

                
END_METHOD

METHOD PRIVATE HandleAliveBit
VAR_INPUT
  LifeSign : BYTE;
END_VAR

VAR_INST
  /// flag that indicates that the 1st cyclce is running
  First : BOOL := TRUE;
END_VAR
                  IF (First AND LifeSign > 0)
THEN
  // init alive value
 _aliveValue := LifeSign;
  // reset first flag
  First := FALSE;
END_IF

_aliveCheck ( IN  := (_aliveValue = LifeSign) , PT := ParCfg.Com.LifeSignTimeOut + ParCfg.Plc.CycleTime);
_alive_R    ( CLK := _aliveBit);
_alive_F    ( CLK := _aliveBit);

IF ( _aliveValue <> LifeSign)
THEN
 _aliveValue := LifeSign;
 _aliveBit   := TRUE;
END_IF

IF (_aliveCheck.Q)
THEN
 _aliveBit := FALSE;
END_IF

IF (_alive_R.Q)
THEN
  // Create log entry
  CreateLogMessage ( Timestamp   := SystemTime,
                     MessageType := MessageType.CMD,
                     Severity    := Severity.INFO,
                     MessageCode := 0,
                     MessageText := 'Data Exchange is running (Alive-Bit)');
END_IF

IF (_alive_F.Q)
THEN
  // Create log entry
  CreateLogMessage ( Timestamp   := SystemTime,
                     MessageType := MessageType.CMD,
                     Severity    := Severity.INFO,
                     MessageCode := 0,
                     MessageText := 'Data Exchange has stopped (Alive-Bit)');
END_IF
                
END_METHOD

METHOD PRIVATE HandleAxesGroup
VAR_IN_OUT
  /// Robot assignment of function
  AxesGroup         : AxesGroup;
  /// ToolData stored on PLC. For more information refer to 5.5.6.3
  ToolData          : ARRAY[*] OF Tool;
  /// LoadData stored on PLC.For more information refer to 5.5.6.4
  FrameData         : ARRAY[*] OF Frame;
  /// LoadData stored on PLC.For more information refer to 5.5.6.4 
  LoadData          : ARRAY[*] OF Load;
  /// Work areas stored on PLC. For more information refer to 5.5.8
  WorkAreas         : ARRAY[*] OF RobotWorkArea;
  /// Software limits stored on PLC
  SWLimits          : SWLimits;
  /// Default dynamics stored on PLC. For more information refer to 5.5.7
  DefaultDynamics   : DefaultDynamics;
  /// Reference dynamics stored on PLC. For more information refer to 5.5.7
  ReferenceDynamics : ReferenceDynamics;  
END_VAR
                  HandleAxesGroupAcyclic       ( AxesGroup         := AxesGroup );
HandleAxesGroupCyclic        ( AxesGroup         := AxesGroup );
HandleAxesGroupCyclicOptional( AxesGroup         := AxesGroup );
HandleAxesGroupMessageLog    ( AxesGroup         := AxesGroup );
HandleAxesGroupParameter     ( AxesGroup         := AxesGroup );
HandleAxesGroupState         ( AxesGroup         := AxesGroup );
HandleAxesGroupSystemData    ( AxesGroup         := AxesGroup, 
	                             ToolData          := ToolData, 
	                             FrameData         := FrameData, 
	                             LoadData          := LoadData, 
	                             WorkAreas         := WorkAreas, 
	                             SWLimits          := SWLimits, 
	                             DefaultDynamics   := DefaultDynamics, 
	                             ReferenceDynamics := ReferenceDynamics);
                
END_METHOD

METHOD PRIVATE HandleAxesGroupAcyclic
VAR_IN_OUT
  /// Robot assignment of function
  AxesGroup : AxesGroup;
END_VAR
                  // Call active command register FB
AxesGroup.Acyclic.ActiveCommandRegister(SystemTime     := SystemTime,
                                        RegisterSize   := MIN( RobotLibraryParameter.ACTIVE_CMD_REGISTER_ENTRIES_MAX, AxesGroup.Parameter.Rob.Parameter.LengthACR),
                                        InternalLogger := AxesGroup.MessageLog, 
                                        ExternalLogger := AxesGroup.MessageLog.ExternalLogger,
                                        LogLevel       := AxesGroup.MessageLog.LogLevel);
                
END_METHOD

METHOD PRIVATE HandleAxesGroupCyclic
VAR_IN_OUT
  /// Robot assignment of function
  AxesGroup : AxesGroup;
END_VAR
                  // set instance AxesGroupID
AxesGroup.Cyclic.PlcToRob.AxesGroupID := AxesGroupID;
// Set Version
AxesGroup.Cyclic.PlcToRob.SRCIVersion := RobotLibraryConstants.SRCIVersion;

AxesGroup.Cyclic.PlcToRob.TelegramLengthPlcToRob := _parCfg.Com.TelegramLengthPlcToRob;
AxesGroup.Cyclic.PlcToRob.TelegramLengthRobToPlc := _parCfg.Com.TelegramLengthRobToPlc;

AxesGroup.Cyclic.PlcToRob.TelegramNumberPlcToRob := PlcOptionalCyclicToUint(AxesGroup.Parameter.Plc.OptionalCyclic);
AxesGroup.Cyclic.PlcToRob.TelegramNumberRobToPlc := RobOptionalCyclicToUint(AxesGroup.Parameter.Rob.OptionalCyclic);

// Set Date + Time
AxesGroup.Cyclic.PlcToRob.ClientDate  := DATE_TO_IEC_DATE(SystemTime.SystemDate);
AxesGroup.Cyclic.PlcToRob.ClientTime  := TIME_TO_IEC_TIME(SystemTime.SystemTime);
                
END_METHOD

METHOD PRIVATE HandleAxesGroupCyclicOptional
VAR_IN_OUT
  /// Robot assignment of function
  AxesGroup : AxesGroup;
END_VAR
                  // PlcToRob {{{
AxesGroup.CyclicOptional.PlcToRob.SubProgramData      .Active := AxesGroup.Parameter.Plc.OptionalCyclic.UseCallSubprogram; 
AxesGroup.CyclicOptional.PlcToRob.CartesianPosition   .Active := AxesGroup.Parameter.Plc.OptionalCyclic.UseCartesianPosition; 
AxesGroup.CyclicOptional.PlcToRob.JointPosition       .Active := AxesGroup.Parameter.Plc.OptionalCyclic.UseJointPosition; 
AxesGroup.CyclicOptional.PlcToRob.Force               .Active := AxesGroup.Parameter.Plc.OptionalCyclic.UseForce; 
AxesGroup.CyclicOptional.PlcToRob.CartesianPositionExt.Active := AxesGroup.Parameter.Plc.OptionalCyclic.UseCartesianPositionExt; 
AxesGroup.CyclicOptional.PlcToRob.JointPositionExt    .Active := AxesGroup.Parameter.Plc.OptionalCyclic.UseJointPositionExt; 
// }}}

// RobToPlc {{{
AxesGroup.CyclicOptional.RobToPlc.SubProgramData      .Active := AxesGroup.Parameter.Rob.OptionalCyclic.UseCallSubprogram; 
AxesGroup.CyclicOptional.RobToPlc.CartesianPosition   .Active := AxesGroup.Parameter.Rob.OptionalCyclic.UseCartesianPosition;    
AxesGroup.CyclicOptional.RobToPlc.JointPosition       .Active := AxesGroup.Parameter.Rob.OptionalCyclic.UseJointPosition;    
AxesGroup.CyclicOptional.RobToPlc.Force               .Active := AxesGroup.Parameter.Rob.OptionalCyclic.UseForce;
AxesGroup.CyclicOptional.RobToPlc.Current             .Active := AxesGroup.Parameter.Rob.OptionalCyclic.UseCurrent;    
AxesGroup.CyclicOptional.RobToPlc.CartesianPositionExt.Active := AxesGroup.Parameter.Rob.OptionalCyclic.UseCartesianPositionExt;    
AxesGroup.CyclicOptional.RobToPlc.JointPositionExt    .Active := AxesGroup.Parameter.Rob.OptionalCyclic.UseJointPositionExt;    
AxesGroup.CyclicOptional.RobToPlc.ForceExt            .Active := AxesGroup.Parameter.Rob.OptionalCyclic.UseForceExt;    
AxesGroup.CyclicOptional.RobToPlc.CurrentExt          .Active := AxesGroup.Parameter.Rob.OptionalCyclic.UseCurrentExt;    
// }}}

                
END_METHOD

METHOD PRIVATE HandleAxesGroupMessageLog
VAR_IN_OUT
  /// Robot assignment of function
  AxesGroup  : AxesGroup;
END_VAR
                  // Set External logger 
AxesGroup.MessageLog.ExternalLogger := ExternalLogger;
AxesGroup.MessageLog.LogLevel       := LogLevel;


IF (AxesGroup.State.GroupReset_R.Q)
THEN
  AxesGroup.MessageLog.DeleteMessages();
  AxesGroup.MessageLog.DeleteSystemLogs();
END_IF
                
END_METHOD

METHOD PRIVATE HandleAxesGroupParameter
VAR_IN_OUT
  /// Robot assignment of function
  AxesGroup : AxesGroup;
END_VAR
                  IF (_exchangeConfiguration.Enabled)
THEN
  AxesGroup.Parameter.Plc.Parameter                           := _parCfg.Plc.Parameter;      
  AxesGroup.Parameter.Plc.OptionalCyclic                      := _parCfg.Plc.OptionalCyclic;
  AxesGroup.Parameter.Rob.OptionalCyclic                      := _parCfg.Rob.OptionalCyclic;
  
  AxesGroup.Parameter.Rob.Parameter.LengthACR                 := _exchangeConfiguration.OutCmd.LengthACR;
  AxesGroup.Parameter.Rob.Parameter.HighestToolIndex          := _exchangeConfiguration.OutCmd.HighestToolIndex;
  AxesGroup.Parameter.Rob.Parameter.HighestFrameIndex         := _exchangeConfiguration.OutCmd.HighestFrameIndex;
  AxesGroup.Parameter.Rob.Parameter.HighestLoadIndex          := _exchangeConfiguration.OutCmd.HighestLoadIndex;
  AxesGroup.Parameter.Rob.Parameter.HighestWorkAreaIndex      := _exchangeConfiguration.OutCmd.HighestWorkAreaIndex;
  AxesGroup.Parameter.Rob.Parameter.DataInSync                := _exchangeConfiguration.OutCmd.DataInSync;
  AxesGroup.Parameter.Rob.Parameter.ChangeIndexTool           := _exchangeConfiguration.OutCmd.ChangeIndexTool;
  AxesGroup.Parameter.Rob.Parameter.ChangeIndexFrame          := _exchangeConfiguration.OutCmd.ChangeIndexFrame;
  AxesGroup.Parameter.Rob.Parameter.ChangeIndexLoad           := _exchangeConfiguration.OutCmd.ChangeIndexLoad;
  AxesGroup.Parameter.Rob.Parameter.ChangeIndexWorkArea       := _exchangeConfiguration.OutCmd.ChangeIndexWorkArea;
  AxesGroup.Parameter.Rob.Parameter.RAWorkingHours            := _exchangeConfiguration.OutCmd.RAWorkingHours;
  AxesGroup.Parameter.Rob.Parameter.BrakeTestRequired         := _exchangeConfiguration.OutCmd.BrakeTestRequired;
  AxesGroup.Parameter.Rob.Parameter.StepModeExactStopActive   := _exchangeConfiguration.OutCmd.StepModeExactStopActive;
  AxesGroup.Parameter.Rob.Parameter.StepModeBlendingActive    := _exchangeConfiguration.OutCmd.StepModeBlendingActive;
  AxesGroup.Parameter.Rob.Parameter.PathAccuracyMode          := _exchangeConfiguration.OutCmd.PathAccuracyMode;
  AxesGroup.Parameter.Rob.Parameter.AvoidSingularity          := _exchangeConfiguration.OutCmd.AvoidSingularity;
  AxesGroup.Parameter.Rob.Parameter.CollisionDetectionEnabled := _exchangeConfiguration.OutCmd.CollisionDetectionEnabled;
  AxesGroup.Parameter.Rob.Parameter.AcceleratingSupported     := _exchangeConfiguration.OutCmd.AcceleratingSupported;
  AxesGroup.Parameter.Rob.Parameter.DecceleratingSupported    := _exchangeConfiguration.OutCmd.DecceleratingSupported;
  AxesGroup.Parameter.Rob.Parameter.ConstantVelocitySupported := _exchangeConfiguration.OutCmd.ConstantVelocitySupported;
  AxesGroup.Parameter.Rob.Parameter.RCWorkingHours            := _exchangeConfiguration.OutCmd.RCWorkingHours;
ELSE
  AxesGroup.Parameter.Plc.Parameter                           := ParCfg.Plc.Parameter;      
  AxesGroup.Parameter.Plc.OptionalCyclic                      := ParCfg.Plc.OptionalCyclic;
  AxesGroup.Parameter.Rob.OptionalCyclic                      := ParCfg.Rob.OptionalCyclic;
END_IF
                
END_METHOD

METHOD PRIVATE HandleAxesGroupState
VAR_IN_OUT
  /// Robot assignment of function
  AxesGroup : AxesGroup;
END_VAR
VAR
  /// internal index for loops
 _idx       : DINT; 
END_VAR
                  AxesGroup.State.AliveOk      := _aliveBit;
AxesGroup.State.Initialized  := Initialized  AND AxesGroup.State.AliveOk;
AxesGroup.State.Synchronized := Synchronized AND AxesGroup.State.AliveOk;
AxesGroup.State.CMDsEnabled  := AxesGroup.State.Initialized OR 
                                AxesGroup.State.Synchronized;

AxesGroup.State.StatusRobotArm  := AxesGroup.Cyclic.RobToPlc.StatusRobotArm;                                
AxesGroup.State.ConfigExchanged := _exchangeConfiguration.Enabled;

AxesGroup.State.UnifiedFrameIndex                    := DINT_TO_USINT( MIN( MIN(AxesGroup.SystemData.FrameDataMax, RobotLibraryParameter.FRAME_MAX     ), _exchangeConfiguration.OutCmd.HighestFrameIndex   ));
AxesGroup.State.UnifiedToolIndex                     := DINT_TO_USINT( MIN( MIN(AxesGroup.SystemData.ToolDataMax , RobotLibraryParameter.TOOL_MAX      ), _exchangeConfiguration.OutCmd.HighestToolIndex    ));
AxesGroup.State.UnifiedLoadIndex                     := DINT_TO_USINT( MIN( MIN(AxesGroup.SystemData.LoadDataMax , RobotLibraryParameter.LOAD_MAX      ), _exchangeConfiguration.OutCmd.HighestLoadIndex    ));
AxesGroup.State.UnifiedWorkAreaIndex                 := DINT_TO_USINT( MIN( MIN(AxesGroup.SystemData.WorkAreasMax, RobotLibraryParameter.WORK_AREAS_MAX), _exchangeConfiguration.OutCmd.HighestWorkAreaIndex));

AxesGroup.State.DataEnableSync                       := _exchangeConfiguration.ParCmd.DataEnableSync;
AxesGroup.State.SyncStateRc.InSync.Frame             := _exchangeConfiguration.OutCmd.DataInSync.FramesInSync;
AxesGroup.State.SyncStateRc.InSync.Tool              := _exchangeConfiguration.OutCmd.DataInSync.ToolsInSync;
AxesGroup.State.SyncStateRc.InSync.Load              := _exchangeConfiguration.OutCmd.DataInSync.LoadsInSync;
AxesGroup.State.SyncStateRc.InSync.WorkArea          := _exchangeConfiguration.OutCmd.DataInSync.WorkAreasInSync;
AxesGroup.State.SyncStateRc.InSync.SwLimits          := _exchangeConfiguration.OutCmd.DataInSync.SoftwareLimitsInSync;
AxesGroup.State.SyncStateRc.InSync.DefaultDynamics   := _exchangeConfiguration.OutCmd.DataInSync.DefaultDynamicsInSync;
AxesGroup.State.SyncStateRc.InSync.ReferenceDynamics := _exchangeConfiguration.OutCmd.DataInSync.ReferenceDynamicsInSync;

AxesGroup.State.SyncStateRc.UnSyncNo.Frame           := _exchangeConfiguration.OutCmd.ChangeIndexFrame;
AxesGroup.State.SyncStateRc.UnSyncNo.Tool            := _exchangeConfiguration.OutCmd.ChangeIndexTool;
AxesGroup.State.SyncStateRc.UnSyncNo.Load            := _exchangeConfiguration.OutCmd.ChangeIndexLoad;
AxesGroup.State.SyncStateRc.UnSyncNo.WorkArea        := _exchangeConfiguration.OutCmd.ChangeIndexWorkArea;

// Update internal data
AxesGroup.State.SystemTime   := SystemTime;
AxesGroup.State.OnlineChange := OnlineChange;
AxesGroup.State.Initialized  := Initialized;

// Create rising and falling edges for Online Change
AxesGroup.State.OnlineChange_R(CLK := OnlineChange);
AxesGroup.State.OnlineChange_F(CLK := OnlineChange);

// Create rising and falling edges for GroupReset
AxesGroup.State.GroupReset_R(CLK := AxesGroup.State.GroupReset);
AxesGroup.State.GroupReset_F(CLK := AxesGroup.State.GroupReset);

// Copy function block results 
AxesGroup.State.RobotData         := _readRobotData.OutCmd;
AxesGroup.State.ConfigurationData := _exchangeConfiguration.OutCmd;
                
END_METHOD

METHOD PRIVATE HandleAxesGroupSystemData
VAR_IN_OUT
  /// Robot assignment of function
  AxesGroup         : AxesGroup;
  /// ToolData stored on PLC. For more information refer to 5.5.6.3
  ToolData          : ARRAY[*] OF Tool;
  /// LoadData stored on PLC.For more information refer to 5.5.6.4
  FrameData         : ARRAY[*] OF Frame;
  /// LoadData stored on PLC.For more information refer to 5.5.6.4 
  LoadData          : ARRAY[*] OF Load;
  /// Work areas stored on PLC. For more information refer to 5.5.8
  WorkAreas         : ARRAY[*] OF RobotWorkArea;
  /// Software limits stored on PLC
  SWLimits          : SWLimits;
  /// Default dynamics stored on PLC. For more information refer to 5.5.7
  DefaultDynamics   : DefaultDynamics;
  /// Reference dynamics stored on PLC. For more information refer to 5.5.7
  ReferenceDynamics : ReferenceDynamics;  
END_VAR
                  // Update ToolData                    
AxesGroup.SystemData.ToolDataPtr       := ToolData;
AxesGroup.SystemData.ToolDataMin       := LOWER_BOUND  (ToolData,1);
AxesGroup.SystemData.ToolDataMax       := UPPER_BOUND  (ToolData,1);
AxesGroup.SystemData.ToolDataCount     := DINT_TO_UDINT(1 + AxesGroup.SystemData.ToolDataMax - AxesGroup.SystemData.ToolDataMin);
                                       
// Update LoadData                    
AxesGroup.SystemData.LoadDataPtr       := LoadData;
AxesGroup.SystemData.LoadDataMin       := LOWER_BOUND  (LoadData,1);                                                    
AxesGroup.SystemData.LoadDataMax       := UPPER_BOUND  (LoadData,1);                                                    
AxesGroup.SystemData.LoadDataCount     := DINT_TO_UDINT(1 + AxesGroup.SystemData.LoadDataMax - AxesGroup.SystemData.LoadDataMin);
                                       
// Update FrameData       
AxesGroup.SystemData.FrameDataPtr      := LoadData;                                                                       
AxesGroup.SystemData.FrameDataMin      := LOWER_BOUND  (LoadData,1);                                                     
AxesGroup.SystemData.FrameDataMax      := UPPER_BOUND  (LoadData,1);                                                     
AxesGroup.SystemData.FrameDataCount    := DINT_TO_UDINT(1 + AxesGroup.SystemData.FrameDataMax - AxesGroup.SystemData.FrameDataMin);

// Update WorkAreas 
AxesGroup.SystemData.WorkAreasPtr      := LoadData;                                                                      
AxesGroup.SystemData.WorkAreasMin      := LOWER_BOUND  (LoadData,1);                                                     
AxesGroup.SystemData.WorkAreasMax      := UPPER_BOUND  (LoadData,1);                                                     
AxesGroup.SystemData.WorkAreasCount    := DINT_TO_UDINT(1 + AxesGroup.SystemData.WorkAreasMax - AxesGroup.SystemData.WorkAreasMin);

// Update SoftwareLimits 
AxesGroup.SystemData.SWLimits          REF= SWLimits;
// Update DefaultDynamics 
AxesGroup.SystemData.DefaultDynamics   REF= DefaultDynamics;
// Update ReferenceDynamics 
AxesGroup.SystemData.ReferenceDynamics REF= ReferenceDynamics;
                
END_METHOD

METHOD PRIVATE HandleInvalidFrames
VAR_IN_OUT
   /// Robot assignment of function
  AxesGroup   : AxesGroup;
    /// Inputs of PLC for communication from RC
  RobotInData : ARRAY[*] OF BYTE;
END_VAR 
VAR
  /// Value of lifesign in header
 _lifeSignHeader    : BYTE;
  /// Value of lifesign in footer
 _lifeSignFooter    : BYTE;
END_VAR
VAR_INST
  /// Timeout for invalid frames counter check
 _invalidFrameCounterCheck_D : TON;
  /// last count of invalid frames
 _lastInvalidFrames          : UDINT;
END_VAR
                  IF ( AxesGroup.Cyclic.RobToPlc.TelegramState = TelegramState.INITIALIZED ) 
THEN
  // Get lifesign values
 _lifeSignHeader := GetHalfeByteHi( RobotInData[ROBOT_IN_DATA_MIN + 1]);
 _lifeSignFooter := GetHalfeByteHi( RobotInData[ROBOT_IN_DATA_MAX + 0]);
END_IF

// Timer for invalid frame(s) message
_invalidFrameCounterCheck_D( IN := TRUE , PT := RobotLibraryParameter.INVALID_FRAMES_CHECK_TIMEOUT);

// Check Frame is valid : 
// ----------------------
IF ( _lifeSignHeader <> _lifeSignFooter )   
THEN
  AxesGroup.State.InvalidFrames := AxesGroup.State.InvalidFrames + 1;
END_IF


// Check timeout for invalid frame message
IF ( _invalidFrameCounterCheck_D.Q )
THEN
  // reset timer
 _invalidFrameCounterCheck_D( IN := FALSE);
  
  // compare invalid frame(s) counter
  IF ( AxesGroup.State.InvalidFrames <> _lastInvalidFrames)
  THEN
    // store last invalid frame(s) counter value
   _lastInvalidFrames := AxesGroup.State.InvalidFrames;
    // Create log entry
    CreateLogMessagePara1 ( Timestamp   := SystemTime,
                            MessageType := MessageType.CMD,
                            Severity    := Severity.WARNING,
                            MessageCode := 0,
                            MessageText := 'Detected invalid frames {1} in total',
                            Para1       :=  UDINT_TO_STRING(AxesGroup.State.InvalidFrames));
  END_IF
END_IF


// Reset invalid frames counter with rising edge of group reset
IF ( AxesGroup.State.GroupReset_R.Q)
THEN
  AxesGroup.State.InvalidFrames := 0;
             _lastInvalidFrames := 0;
 
  // Create log entry
  CreateLogMessage ( Timestamp   := SystemTime,
                     MessageType := MessageType.CMD,
                     Severity    := Severity.INFO,
                     MessageCode := 0,
                     MessageText := 'Reset invalid frames counter by executing GroupReset');
END_IF
                
END_METHOD

METHOD PRIVATE HandleLifeSign
VAR_IN_OUT
  /// Robot assignment of function
  AxesGroup    : AxesGroup;
END_VAR 
VAR_INST
  /// flag for 1st cycle
 _first : BOOL := TRUE;
END_VAR
                  IF ( _first ) OR ( NOT Enable ) 
THEN
  // init LifeSign 
  AxesGroup.Cyclic.PlcToRob.LifeSign := 0;
  // reset first flag
 _first := FALSE;
  // prevent inc LifeSign in the 1st cycle (Code below)
  RETURN;
END_IF


AxesGroup.Cyclic.PlcToRob.LifeSign := AxesGroup.Cyclic.PlcToRob.LifeSign + 1;
  
IF ( AxesGroup.Cyclic.PlcToRob.LifeSign > 15 )
THEN
  AxesGroup.Cyclic.PlcToRob.LifeSign := 1; // 0 is only in the very 1st cycle to indicate the system start in logging
END_IF


IF ( Enable ) AND ( _alive_F.Q ) 
THEN
  // Reset initialized flag
  Initialized := FALSE;
  // Reset Synchronized flag
  Synchronized := FALSE;
  
  // Set error 
  SetError( ErrorID := RobotLibraryErrorIdEnum.ERR_CONNECTION_LOST, Overwrite := TRUE );  
  // Create log entry
  CreateLogMessage ( Timestamp   := SystemTime,
                     MessageType := MessageType.CMD,
                     Severity    := Severity.FATAL_ERROR,
                     MessageCode := 0,
                     MessageText := 'LifeSign timeout -> Reinitialization required !');
END_IF

// Reset connection lost error
IF ( NOT Enable ) AND ( _aliveBit ) AND ( ErrorID = RobotLibraryErrorIdEnum.ERR_CONNECTION_LOST )
THEN
  ErrorID := 0;
END_IF
                
END_METHOD

METHOD HandleLogMessagesAck
VAR_IN_OUT
   /// Robot assignment of function
  AxesGroup : AxesGroup;
END_VAR
                  IF ( _readMessages.Enabled )  
THEN
  // Set Message ID as Acknowlege ID  
 _readMessages.ParCmd.MsgID := _readMessages.OutCmd.MsgId;  
ELSE
  // Reset Acknowlege ID  
 _readMessages.ParCmd.MsgID := 0;
END_IF 



(*

IF (( _readMessages.Enabled           ) AND 
    ( _readMessages.OutCmd.MsgId > 0  ))  
THEN
  // Check if message has been entered into the message log ?   
  IF ( AxesGroup.MessageLog.CheckMessageCodePresent(_readMessages.OutCmd.ErrorCode ))
  THEN
    // Set Message ID as Acknowlege ID  
   _readMessages.ParCmd.MsgID := _readMessages.OutCmd.MsgId;  
	END_IF    
END_IF

*)
                
END_METHOD

METHOD PRIVATE HandleSeqAck
VAR_IN_OUT
   /// Robot assignment of function
  AxesGroup    : AxesGroup;
END_VAR 
VAR
  /// internal index for loops
 _idx : DINT;
END_VAR
                  FOR _idx := 0 TO  AxesGroup.State.SequenceCountSend 
DO
  AxesGroup.State.CurrentAck[_idx] := Telegram.RobToPlc.Sequence[_idx].Header.SEQ_ACK;
  
  IF (NOT Enable)
  THEN
    AxesGroup.State.CurrentSEQ[0] := 0;
    AxesGroup.State.CurrentSEQ[1] := 0;
  END_IF  
  
  // Check Seq/Ack : 
  // ----------------------
  IF ( AxesGroup.State.CurrentAck[_idx] = AxesGroup.State.CurrentSEQ[_idx] ) 
  THEN
    AxesGroup.State.CurrentSEQ[_idx] := MAX(AxesGroup.State.CurrentSEQ[0],AxesGroup.State.CurrentSEQ[1]) +1;

    IF (AxesGroup.State.CurrentSEQ[_idx] >= 255) {warning 'ToDo: Test for Yaskawa'}
    THEN
      AxesGroup.State.CurrentSEQ[_idx] := 0;
		END_IF
    
    AxesGroup.State.NewSEQ[_idx] := TRUE;
  END_IF  
END_FOR
                
END_METHOD

METHOD PRIVATE HandleSync
VAR_IN_OUT
   /// Robot assignment of function
  AxesGroup : AxesGroup;
  /// ToolData stored on PLC.For more information refer to 5.5.6.4
  ToolData          : ARRAY[*] OF Tool;
  /// LoadData stored on PLC.For more information refer to 5.5.6.4
  FrameData         : ARRAY[*] OF Frame;
  /// LoadData stored on PLC.For more information refer to 5.5.6.4
  LoadData          : ARRAY[*] OF Load;
  /// Work areas stored on PLC. For more information refer to 5.5.8
  WorkAreas         : ARRAY[*] OF RobotWorkArea;
  /// Software limits stored on PLC
  SWLimits          : SWLimits;
  /// Default dynamics stored on PLC. For more information refer to 5.5.7
  DefaultDynamics   : DefaultDynamics;
  /// Reference dynamics stored on PLC. For more information refer to 5.5.7
  ReferenceDynamics : ReferenceDynamics;
END_VAR 

VAR
  /// flag that indicates at least any iten has enabled synchronisation
 _dataEnableSyncAny        : BOOL; 
  /// flag that indicates that the frame datas are synchronized or deactivated 
 _inSyncFrameOk            : BOOL;      
  /// flag that indicates that the tool datas are synchronized or deactivated 
 _inSyncToolOk             : BOOL;     
  /// flag that indicates that the load datas are synchronized or deactivated 
 _inSyncLoadOk             : BOOL;     
  /// flag that indicates that the work areas are synchronized or deactivated 
 _inSyncWorkAreaOk         : BOOL;
  /// flag that indicates that the SW limits are synchronized or deactivated 
 _inSyncSwLimitsOk         : BOOL;
  /// flag that indicates that the default dynamice are synchronized or deactivated 
 _inSyncDefaultDynamicOk   : BOOL;
  /// flag that indicates that the reference dynamice are synchronized or deactivated 
 _InSyncReferenceDynamicOk : BOOL;
END_VAR
                  HandleSyncToolData              ( AxesGroup := AxesGroup, ToolData          := ToolData);
HandleSyncFrameData             ( AxesGroup := AxesGroup, FrameData         := FrameData);
HandleSyncLoadData              ( AxesGroup := AxesGroup, LoadData          := LoadData);
HandleSyncRobotDefaultDynamics  ( AxesGroup := AxesGroup, DefaultDynamics   := DefaultDynamics);
HandleSyncRobotReferenceDynamics( AxesGroup := AxesGroup, ReferenceDynamics := ReferenceDynamics);
HandleSyncRobotSWLimits         ( AxesGroup := AxesGroup, SwLimits          := SwLimits);
HandleSyncToolData              ( AxesGroup := AxesGroup, ToolData          := ToolData);
HandleSyncWorkArea              ( AxesGroup := AxesGroup, WorkAreas         := WorkAreas);


// check any synchronisation activated ?
_dataEnableSyncAny :=        ((     AxesGroup.State.DataEnableSync.EnableSyncFrame             )  OR
                              (     AxesGroup.State.DataEnableSync.EnableSyncTool              )  OR
                              (     AxesGroup.State.DataEnableSync.EnableSyncLoad              )  OR
                              (     AxesGroup.State.DataEnableSync.EnableSyncWorkArea          )  OR
                              (     AxesGroup.State.DataEnableSync.EnableSyncSWLimits          )  OR
                              (     AxesGroup.State.DataEnableSync.EnableSyncDefaultDynamics   )  OR
                              (     AxesGroup.State.DataEnableSync.EnableSyncReferenceDynamics ));
                       
_inSyncFrameOk :=            ((     AxesGroup.State.SyncStatePlc     .InSync.Frame             )  AND 
                              (     AxesGroup.State.SyncStateRc      .InSync.Frame             )) OR
                              ( NOT AxesGroup.State.DataEnableSync.EnableSyncFrame             );
                                                                                       
_inSyncToolOk :=             ((     AxesGroup.State.SyncStatePlc     .InSync.Tool              )  AND 
                              (     AxesGroup.State.SyncStateRc      .InSync.Tool              )) OR
                              ( NOT AxesGroup.State.DataEnableSync.EnableSyncTool              ); 
                                                                                           
_inSyncLoadOk :=             ((     AxesGroup.State.SyncStatePlc     .InSync.Load              )  AND 
                              (     AxesGroup.State.SyncStateRc      .InSync.Load              )) OR
                              ( NOT AxesGroup.State.DataEnableSync.EnableSyncLoad              ); 
                                                                                           
_inSyncWorkAreaOk :=         ((     AxesGroup.State.SyncStatePlc     .InSync.WorkArea          )  AND 
                              (     AxesGroup.State.SyncStateRc      .InSync.WorkArea          )) OR
                              ( NOT AxesGroup.State.DataEnableSync.EnableSyncWorkArea          ); 
                                                                                           
_inSyncSwLimitsOk :=         ((     AxesGroup.State.SyncStatePlc    .InSync.SwLimits           )  AND 
                              (     AxesGroup.State.SyncStateRc      .InSync.SwLimits          )) OR
                              ( NOT AxesGroup.State.DataEnableSync.EnableSyncSwLimits          ); 
                       
_inSyncDefaultDynamicOk :=   ((     AxesGroup.State.SyncStatePlc     .InSync.DefaultDynamics   )  AND 
                              (     AxesGroup.State.SyncStateRc      .InSync.DefaultDynamics   )) OR
                              ( NOT AxesGroup.State.DataEnableSync.EnableSyncDefaultDynamics   ); 

_inSyncReferenceDynamicOk := ((     AxesGroup.State.SyncStatePlc     .InSync.ReferenceDynamics )  AND 
                              (     AxesGroup.State.SyncStateRc      .InSync.ReferenceDynamics )) OR
                              ( NOT AxesGroup.State.DataEnableSync.EnableSyncReferenceDynamics ); 
                       
                       
Synchronized := (( _inSyncFrameOk            ) AND      
                 ( _inSyncToolOk             ) AND    
                 ( _inSyncLoadOk             ) AND     
                 ( _inSyncWorkAreaOk         ) AND     
                 ( _inSyncSwLimitsOk         ) AND     
                 ( _inSyncDefaultDynamicOk   ) AND     
                 ( _InSyncReferenceDynamicOk ) AND            
                 ( _dataEnableSyncAny        ));                                                                                                                                                      


// Update exchange configuration parameter
_exchangeConfiguration.ParCmd.DataInSync.FramesInSync            := AxesGroup.State.SyncStatePlc.InSync.Frame;                // OR ( NOT AxesGroup.State.DataEnableSync.EnableSyncFrame            );
_exchangeConfiguration.ParCmd.DataInSync.ToolsInSync             := AxesGroup.State.SyncStatePlc.InSync.Tool;                 // OR ( NOT AxesGroup.State.DataEnableSync.EnableSyncTool             );
_exchangeConfiguration.ParCmd.DataInSync.LoadsInSync             := AxesGroup.State.SyncStatePlc.InSync.Load;                 // OR ( NOT AxesGroup.State.DataEnableSync.EnableSyncLoad             );
_exchangeConfiguration.ParCmd.DataInSync.WorkAreasInSync         := AxesGroup.State.SyncStatePlc.InSync.WorkArea;             // OR ( NOT AxesGroup.State.DataEnableSync.EnableSyncWorkArea         );
_exchangeConfiguration.ParCmd.DataInSync.SoftwareLimitsInSync    := AxesGroup.State.SyncStatePlc.InSync.SwLimits;             // OR ( NOT AxesGroup.State.DataEnableSync.EnableSyncSWLimits         );
_exchangeConfiguration.ParCmd.DataInSync.DefaultDynamicsInSync   := AxesGroup.State.SyncStatePlc.InSync.DefaultDynamics;      // OR ( NOT AxesGroup.State.DataEnableSync.EnableSyncDefaultDynamics  );
_exchangeConfiguration.ParCmd.DataInSync.ReferenceDynamicsInSync := AxesGroup.State.SyncStatePlc.InSync.ReferenceDynamics;    // OR ( NOT AxesGroup.State.DataEnableSync.EnableSyncReferenceDynamics);
                
END_METHOD

METHOD PRIVATE HandleSyncFrameData
VAR_IN_OUT
   /// Robot assignment of function
  AxesGroup : AxesGroup;
  /// FrameData stored on PLC.For more information refer to 5.5.6.4
  FrameData : ARRAY[*] OF Frame;
END_VAR 

VAR
  /// Internal step counter name
 _stepName        : STRING;    
  /// Internal reference to step counter
 _rStep           : REFERENCE TO DINT;
  /// Internal reference to timer
 _rTimer          : REFERENCE TO TON;
  /// Internal reference to timeout
 _rTimeout        : REFERENCE TO TIME; 
  /// Internal reference to synchroniztion index
 _rSyncIdx        : REFERENCE TO USINT;
  /// internal bit for condition found
 _found           : BOOL;
  /// empty data set to reset all DataChanged bits
 _dataChangedNone : AxesGroupStateDataChanged;
  /// internal index for loops
 _idx             : DINT;
END_VAR
                  // Set internal references 
_stepName      :=   '_stepSyncFrameData = ';
_rStep       REF=    _stepSyncFrameData;
_rTimer      REF=   _timerSyncFrameData;
_rTimeout    REF= _timeoutSyncFrameData;
_rSyncIdx    REF=     _syncIdxFrameData;


CASE _rStep
OF    
  0: // Check initialisation configured ?
     IF (( _parCfg.PLC.Parameter.SynchronizationModes.Frame[SyncTime.DURING_START_UP] = SyncMode.NO_SYNCHRONIZATION ) AND
         ( _parCfg.PLC.Parameter.SynchronizationModes.Frame[SyncTime. AFTER_START_UP] = SyncMode.NO_SYNCHRONIZATION ))
     THEN
       RETURN;
     END_IF

     // Check More Data on RC than on PLC -> Synchronization not possible
     IF (AxesGroup.State.ConfigurationData.HighestFrameIndex > AxesGroup.SystemData.FrameDataCount)
     THEN
       SetError( ErrorID := RobotLibraryErrorIdEnum.ERR_SYNC_FRAME_COUNT_RC_HIGHER_THAN_PLC, Overwrite := FALSE);
       RETURN;
		 END_IF
     
     // wait for initialisation done
     IF  ((     AxesGroup.State.RobotData.RCSupportedFunctions. ReadFrameData ) AND
          (     AxesGroup.State.RobotData.RCSupportedFunctions.WriteFrameData ) AND
          (     AxesGroup.State.Initialized                                   ) AND 
          ( NOT Error                                                         ))  
     THEN
       // Check PLC frames < RC frames and SyncFrame enabled ?    
       IF (( AxesGroup.State.DataEnableSync.EnableSyncFrame      = TRUE                              )  AND
           ( AxesGroup.Parameter.Rob.Parameter.HighestFrameIndex > AxesGroup.SystemData.FrameDataMax ))        
       THEN
         SetWarning( WarningID := RobotLibraryWarningIdEnum.WARN_FRAME_DATA_ARRAY_TOO_SHORT, Overwrite := TRUE);
       END_IF

       // Create log entry
       CreateLogMessagePara1 ( Timestamp   := SystemTime,
                               MessageType := MessageType.CMD,
                               Severity    := Severity.DEBUG,
                               MessageCode := 0,
                               MessageText := 'SyncFrameData: Start initial reading of FrameData from RC',
                               Para1       :=  '');
       
       // init frame number
      _rSyncIdx := DINT_TO_USINT(AxesGroup.SystemData.FrameDataMin);
       // init count of unsynchronized elements
       AxesGroup.State.SyncStatePlc.UnSyncNo.Frame := 0;
       // set timeout
       SetTimeout(PT := _rTimeout, rTimer := _rTimer);
       // inc step counter
      _rStep := _rStep + 1;
     END_IF     

     
     // Start read FrameData
  1: IF (( NOT _readFrameData.Busy  ) AND 
         ( NOT _readFrameData.Error ) AND
         ( NOT _readFrameData.Done  ))
     THEN
       // set command parameter
      _readFrameData.ParCmd.FrameNo := _rSyncIdx;      
       // execute command
      _readFrameData.Execute := TRUE;
       // set timeout
       SetTimeout(PT := _rTimeout, rTimer := _rTimer);
       // inc step counter
      _rStep := _rStep + 1;
     ELSE
       // check error ? 
       IF ( _readFrameData.Error )
       THEN
         SetWarning ( WarningID := RobotLibraryWarningIdEnum.WARN_FRAME_SYNC_FAILED_BY_ERROR_OF_READ_OR_WRITE_CMD, Overwrite := FALSE);           
       END_IF  
       
       // timeout exceeded ? 
       IF (CheckTimeout(_rTimer) = RobotLibraryConstants.OK)
       THEN
         ErrorAddTxt := CONCAT(_stepName, DINT_TO_STRING(_rStep));
         SetError( ErrorID := RobotLibraryErrorIdEnum.ERR_TIMEOUT_CMD, Overwrite := FALSE);
       END_IF
     END_IF
 
     
     // Wait Framedata read
  2: IF (( NOT _readFrameData.Busy  ) AND
         ( NOT _readFrameData.Error ) AND
         (     _readFrameData.Done  ))
     THEN
       // reset execution
      _readFrameData.Execute := FALSE;
       // set available bit
      _frameData[_rSyncIdx].Available := TRUE; 
       FrameData[_rSyncIdx].Available := TRUE;      
       // Copy data
      _frameData[_rSyncIdx].Data := _readFrameData.OutCmd.FrameData;

       // Check frame data is equal ? 
       IF ( NOT IsFrameDataEqual( Data1 := _frameData[_rSyncIdx].Data, Data2 := FrameData[_rSyncIdx].Data, IgnoreTimestamp := TRUE))
       THEN
         // Reset plc in sync flag
         AxesGroup.State.SyncStatePlc.InSync.Frame := FALSE;
         // Set data changed flag
         AxesGroup.State.DataChanged.Frame[_rSyncIdx] := TRUE;
         // inc count of unsynchronised plc frames
         AxesGroup.State.SyncStatePlc.UnSyncNo.Frame := AxesGroup.State.SyncStatePlc.UnSyncNo.Frame + 1;
        
         // Create log entry
         CreateLogMessagePara1 ( Timestamp   := SystemTime,
                                 MessageType := MessageType.CMD,
                                 Severity    := Severity.DEBUG,
                                 MessageCode := 0,
                                 MessageText := 'SyncFrameData: Detected a difference in Frame[{1}] between PLC and RC',
                                 Para1       :=  DINT_TO_STRING(_rSyncIdx));
        
        
         // Check synchronisation is enabled ? 
         IF ( NOT AxesGroup.State.DataEnableSync.EnableSyncFrame )
         THEN
           SetInfo( InfoID := RobotLibraryInfoIdEnum.INFO_SYNC_FRAME_DATA_DISABLED, Overwrite := FALSE);
				 END_IF
         
         // Check user interaction needed ?  
         IF ( AxesGroup.Parameter.PLC.Parameter.SyncUserInteraction.Frame )
         THEN
           SetWarning( WarningID := RobotLibraryWarningIdEnum.WARN_FRAME_NUMBER_SYNC_ERROR, Overwrite := FALSE );                    
				 END_IF
			 END_IF
             
       // Check all frames read ? 
       IF ( _rSyncIdx < AxesGroup.State.UnifiedFrameIndex )
       THEN
         // set timeout
         SetTimeout(PT := _rTimeout, rTimer := _rTimer);
         // inc frame index
        _rSyncIdx := _rSyncIdx + 1;
         // dec step counter
        _rStep := _rStep - 1;
       ELSE
         // set timeout
         SetTimeout(PT := _rTimeout, rTimer := _rTimer);
         // inc step counter
        _rStep := _rStep + 1;           
       END_IF
     ELSE
       // check error ? 
       IF (_readFrameData.Error)
       THEN
         // Set warning
         SetWarning( WarningID := RobotLibraryWarningIdEnum.WARN_FRAME_SYNC_FAILED_BY_ERROR_OF_READ_OR_WRITE_CMD, Overwrite := TRUE);                    
         // reset available bit
         FrameData[_rSyncIdx].Available := FALSE;
        _frameData[_rSyncIdx].Available := FALSE;
       END_IF  
       
       // timeout exceeded ? 
       IF (CheckTimeout(_rTimer) = RobotLibraryConstants.OK)
       THEN
         ErrorAddTxt := CONCAT(_stepName, DINT_TO_STRING(_rStep));
         SetError( ErrorID := RobotLibraryErrorIdEnum.ERR_TIMEOUT_CMD, Overwrite := FALSE);
       END_IF
     END_IF
     
     
     // Check synchronisation state ? 
  3: IF (( AxesGroup.State.SyncStatePlc.UnSyncNo.Frame                                            = 0                           ) OR 
         ( AxesGroup.Parameter.Plc.Parameter.SynchronizationModes.Frame[SyncTime.DURING_START_UP] = SyncMode.NO_SYNCHRONIZATION ))
     THEN
       // Update bit for data in sync
       AxesGroup.State.SyncStatePlc.InSync.Frame := (AxesGroup.State.SyncStatePlc.UnSyncNo.Frame = 0);
       // set timeout
       SetTimeout(PT := _rTimeout, rTimer := _rTimer);
       // inc step counter
      _rStep := 10; // -> jump to after startup
            
       // Create log entry
       CreateLogMessagePara1 ( Timestamp   := SystemTime,
                               MessageType := MessageType.CMD,
                               Severity    := Severity.DEBUG,
                               MessageCode := 0,
                               MessageText := 'SyncFrameData: Synchronization Startup Phase done',
                               Para1       :=  '' );      
     ELSE 
       // Check user interaction needed ? 
       IF ( NOT AxesGroup.Parameter.PLC.Parameter.SyncUserInteraction.Frame )
       THEN
         CASE AxesGroup.Parameter.Plc.Parameter.SynchronizationModes.Frame[SyncTime.DURING_START_UP] OF

           SyncMode.SERVER_TO_CLIENT : 

             FOR _idx := AxesGroup.SystemData.FrameDataMin TO AxesGroup.SystemData.FrameDataMax
             DO
               // Overwrite PLC data with RC data
               FrameData[_idx] := _frameData[_idx];            
						 END_FOR
      
             // Reset data changed flags
             AxesGroup.State.DataChanged.Frame := _dataChangedNone.Frame;
             // Reset Synchronizing flag
             AxesGroup.State.Synchronizing.Frame := FALSE;
             // Set plc in sync flag
             AxesGroup.State.SyncStatePlc.InSync.Frame := TRUE;
             // Reset count of unsynchronised plc frames
             AxesGroup.State.SyncStatePlc.UnSyncNo.Frame := 0;            
             // set timeout
             SetTimeout(PT := _rTimeout, rTimer := _rTimer);
             // inc step counter
            _rStep := 10; // -> jump to after startup         

            // Create log entry
            CreateLogMessagePara3 ( Timestamp   := SystemTime,
                                    MessageType := MessageType.CMD,
                                    Severity    := Severity.DEBUG,
                                    MessageCode := 0,
                                    MessageText := 'SyncFrameData: Synchronization of Frames triggered by StartUp-Compare, SyncMode = {2}, SyncTime = {3}, SyncDirection = RC -> PLC',
                                    Para1       :=  DINT_TO_STRING(_rSyncIdx),
                                    Para2       :=  SYNC_MODE_TO_STRING(AxesGroup.Parameter.Plc.Parameter.SynchronizationModes.Frame[SyncTime.DURING_START_UP]),
                                    Para3       :=  SYNC_TIME_TO_STRING(SyncTime.DURING_START_UP));
            // Create log entry
            CreateLogMessagePara1 ( Timestamp   := SystemTime,
                                    MessageType := MessageType.CMD,
                                    Severity    := Severity.DEBUG,
                                    MessageCode := 0,
                                    MessageText := 'SyncFrameData: Applied the initial read frame data from RC',
                                    Para1       :=  '' );

				   SyncMode.CLIENT_TO_SERVER : ;

             // Check conflicts to solve ? 
             FOR _rSyncIdx := 0 TO AxesGroup.State.UnifiedFrameIndex
             DO
               IF ( AxesGroup.State.DataChanged.Frame[_rSyncIdx] )
               THEN
                _found := TRUE;
                 EXIT;
		  			   END_IF
             END_FOR
           
             IF ( _found ) 
             THEN
               // Reset plc in sync flag
               AxesGroup.State.SyncStatePlc.InSync.Frame := FALSE;
               // Set Synchronizing flag
               AxesGroup.State.Synchronizing.Frame := TRUE;
               // set timeout
               SetTimeout(PT := _rTimeout, rTimer := _rTimer);
               // inc step counter
              _rStep := _rStep +1; // -> write PLC data to RC                  
               // Create log entry
               CreateLogMessagePara3 ( Timestamp   := SystemTime,
                                       MessageType := MessageType.CMD,
                                       Severity    := Severity.DEBUG,
                                       MessageCode := 0,
                                       MessageText := 'SyncFrameData: Synchronization of Frame[{1}] triggered by StartUp-Compare, SyncMode = {2}, SyncTime = {3}, SyncDirection = PLC -> RC',
                                       Para1       :=  DINT_TO_STRING(_rSyncIdx),
                                       Para2       :=  SYNC_MODE_TO_STRING(AxesGroup.Parameter.Plc.Parameter.SynchronizationModes.Frame[SyncTime.DURING_START_UP]),
                                       Para3       :=  SYNC_TIME_TO_STRING(SyncTime.DURING_START_UP));
             ELSE
               // Reset data changed flags
               AxesGroup.State.DataChanged.Frame := _dataChangedNone.Frame;
               // Reset Synchronizing flag
               AxesGroup.State.Synchronizing.Frame := FALSE;
               // Set plc in sync flag
               AxesGroup.State.SyncStatePlc.InSync.Frame := TRUE;
               // Reset count of unsynchronised frames
               AxesGroup.State.SyncStatePlc.UnSyncNo.Frame := 0;
               // set timeout
               SetTimeout(PT := _rTimeout, rTimer := _rTimer);
               // inc step counter
              _rStep := 10; // -> jump to after startup                  
				     END_IF
         ELSE
           // invalid sync mode for startup
           SetError( ErrorID := RobotLibraryErrorIdEnum.ERR_SYNC_MODE_INVALID, Overwrite := TRUE );
 	       END_CASE
       END_IF
     END_IF  

     
     // Start write frame data  
  4: IF (( NOT _writeFrameData.Busy  ) AND 
         ( NOT _writeFrameData.Error ))
     THEN
       // set command parameter
      _writeFrameData.ParCmd.FrameNo   := _rSyncIdx;      
      _writeFrameData.ParCmd.FrameData :=  FrameData[_rSyncIdx].Data;
       // execute command
      _writeFrameData.Execute := TRUE;
       // set timeout
       SetTimeout(PT := _rTimeout, rTimer := _rTimer);
       // inc step counter
      _rStep := _rStep + 1;
     ELSE
       // check error ? 
       IF (_writeFrameData.Error)
       THEN
         ErrorID     := _writeFrameData.ErrorID;
         ErrorAddTxt := _writeFrameData.ErrorAddTxt;;
       END_IF  
       
       // timeout exceeded ? 
       IF (CheckTimeout(_rTimer) = RobotLibraryConstants.OK)
       THEN
         ErrorAddTxt := CONCAT(_stepName, DINT_TO_STRING(_rStep));
         SetError( ErrorID := RobotLibraryErrorIdEnum.ERR_TIMEOUT_CMD, Overwrite := FALSE);
       END_IF
     END_IF
 
     
     // Wait frame data written ?   
  5: IF (( NOT _writeFrameData.Busy  ) AND
         ( NOT _writeFrameData.Error ) AND
         (     _writeFrameData.Done  ))
     THEN
       // execute command
      _writeFrameData.Execute := FALSE;
       // apply frame data to internal frame data
      _frameData[_rSyncIdx] := FrameData[_rSyncIdx];
       // reset data changed bit 
       AxesGroup.State.DataChanged.Frame[_rSyncIdx] := FALSE;
       // dec count of unsynchronised frames
       AxesGroup.State.SyncStatePlc.UnSyncNo.Frame := AxesGroup.State.SyncStatePlc.UnSyncNo.Frame - 1;
       // set timeout        
       SetTimeout(PT := _rTimeout, rTimer := _rTimer);
       // dec step counter
      _rStep := _rStep - 2; 
     ELSE
       // check error ? 
       IF (_writeFrameData.Error)
       THEN
         SetWarning( WarningID := RobotLibraryWarningIdEnum.WARN_FRAME_SYNC_FAILED_BY_ERROR_OF_READ_OR_WRITE_CMD, Overwrite := TRUE);           
       END_IF  
       
       // timeout exceeded ? 
       IF (CheckTimeout(_rTimer) = RobotLibraryConstants.OK)
       THEN
         ErrorAddTxt := CONCAT(_stepName, DINT_TO_STRING(_rStep));
         SetError( ErrorID := RobotLibraryErrorIdEnum.ERR_TIMEOUT_CMD, Overwrite := FALSE);
       END_IF
     END_IF

     
  // --------------------------------------------
  // SyncMode after startup : 
  // --------------------------------------------
         
  10 : // check synchronisation active ? 
       IF ( AxesGroup.Parameter.Plc.Parameter.SynchronizationModes.Frame[SyncTime.AFTER_START_UP] = SyncMode.NO_SYNCHRONIZATION)
       THEN
         RETURN;
       END_IF

       // reset count of unsynchronised frames
       AxesGroup.State.SyncStatePlc.UnSyncNo.Frame := 0;

       // Check all frame datas
       FOR _rSyncIdx := 0 TO AxesGroup.State.UnifiedFrameIndex
       DO
         // compare frame data
         AxesGroup.State.DataChanged.Frame[_rSyncIdx] := NOT IsFrameDataEqual( Data1 := FrameData[_rSyncIdx].Data, Data2 := _frameData[_rSyncIdx].Data, IgnoreTimestamp := FALSE);

         // Check Frame data changed ? 
         IF (AxesGroup.State.DataChanged.Frame[_rSyncIdx])
         THEN
           // inc count of unsynchronised plc frames
           AxesGroup.State.SyncStatePlc.UnSyncNo.Frame := AxesGroup.State.SyncStatePlc.UnSyncNo.Frame + 1;
           // Create log entry
           CreateLogMessagePara2 ( Timestamp   := SystemTime,
                                   MessageType := MessageType.CMD,
                                   Severity    := Severity.DEBUG,
                                   MessageCode := 0,
                                   MessageText := 'SyncFrameData: Detected a local change of Frame[{1}] on PLC, SyncTime = {2}',
                                   Para1       :=  DINT_TO_STRING(_rSyncIdx),    
                                   Para2       :=  SYNC_TIME_TO_STRING(SyncTime.AFTER_START_UP));       
				 END_IF

         // Update plc in sync flag
         AxesGroup.State.SyncStatePlc.InSync.Frame := (AxesGroup.State.SyncStatePlc.UnSyncNo.Frame = 0); 
	     END_FOR

       // Check synchronization is needed ? 
       IF ( NOT AxesGroup.State.SyncStatePlc.InSync.Frame ) XOR  
          ( NOT AxesGroup.State.SyncStateRc .InSync.Frame )
       THEN
         CASE AxesGroup.Parameter.Plc.Parameter.SynchronizationModes.Frame[SyncTime.AFTER_START_UP] 
         OF         
           // NO_SYNCHRONIZATION
           SyncMode.NO_SYNCHRONIZATION : ; // no further action 
           
           // CLIENT_TO_SERVER
           SyncMode.CLIENT_TO_SERVER :
             // set timeout
             SetTimeout(PT := _rTimeout, rTimer := _rTimer);
             // inc step counter
            _rStep := 11;
  
           // SERVER_TO_CLIENT
           SyncMode.SERVER_TO_CLIENT :
             // set timeout
             SetTimeout(PT := _rTimeout, rTimer := _rTimer);
             // inc step counter
            _rStep := 12;
  
           // AUTOMATIC
           SyncMode.AUTOMATIC : 
             // set timeout
             SetTimeout(PT := _rTimeout, rTimer := _rTimer);
             // inc step counter
            _rStep := 13;
         END_CASE
       ELSE
         // datas changeḍ on both sides ? -> Warning 
         IF (( NOT AxesGroup.State.SyncStatePlc.InSync.Frame ) AND  
             ( NOT AxesGroup.State.SyncStateRc .InSync.Frame ))
         THEN
           SetWarning( WarningID := RobotLibraryWarningIdEnum.WARN_FRAME_SYNC_BOTH_SIDES_CHANGED, Overwrite := TRUE);
         END_IF
       END_IF


  // ------------------------------------------
  // SyncMode : CLIENT_TO_SERVER 
  // ------------------------------------------  
  11 : // Conflict triggerd by PLC ?  
       IF ( NOT AxesGroup.State.SyncStatePlc.InSync.Frame )
       THEN
         // search for changed index  
         FOR _rSyncIdx := 0 TO AxesGroup.State.UnifiedFrameIndex
         DO
           IF ( AxesGroup.State.DataChanged.Frame[_rSyncIdx] )
           THEN
             // set timeout
             SetTimeout(PT := _rTimeout, rTimer := _rTimer);
             // inc step counter
            _rStep := 30; // -> write PLC data to RC                  
             EXIT;             
					 END_IF
         END_FOR
         
         // Create log entry
         CreateLogMessagePara3 ( Timestamp   := SystemTime,
                                 MessageType := MessageType.CMD,
                                 Severity    := Severity.DEBUG,
                                 MessageCode := 0,
                                 MessageText := 'SyncFrameData: Synchronization of Frame[{1}] triggered by PLC, SyncMode = {2}, SyncTime = {3}, SyncDirection = PLC -> RC',
                                 Para1       :=  DINT_TO_STRING(_rSyncIdx),
                                 Para2       :=  SYNC_MODE_TO_STRING(AxesGroup.Parameter.Plc.Parameter.SynchronizationModes.Frame[SyncTime.AFTER_START_UP]),
                                 Para3       :=  SYNC_TIME_TO_STRING(SyncTime.AFTER_START_UP));
                                 RETURN;
       END_IF
   
       // Conflict triggered by RC ?
       IF ( NOT AxesGroup.State.SyncStateRc.InSync.Frame )
       THEN
         // get changed index 
        _rSyncIdx := LIMIT(0, AxesGroup.State.SyncStateRc.UnSyncNo.Frame, AxesGroup.State.UnifiedFrameIndex);
         // set timeout
         SetTimeout(PT := _rTimeout, rTimer := _rTimer);
         // inc step counter
        _rStep := 30; // -> write PLC data to RC

         // Create log entry
         CreateLogMessagePara3 ( Timestamp   := SystemTime,
                                 MessageType := MessageType.CMD,
                                 Severity    := Severity.DEBUG,
                                 MessageCode := 0,
                                 MessageText := 'SyncFrameData: Synchronization of Frame[{1}] triggered by RC, SyncMode = {2}, SyncTime = {3}, SyncDirection = PLC -> RC',
                                 Para1       :=  DINT_TO_STRING(_rSyncIdx),
                                 Para2       :=  SYNC_MODE_TO_STRING(AxesGroup.Parameter.Plc.Parameter.SynchronizationModes.Frame[SyncTime.AFTER_START_UP]),
                                 Para3       :=  SYNC_TIME_TO_STRING(SyncTime.AFTER_START_UP));
                                 RETURN;
			 END_IF
       
       // set timeout
       SetTimeout(PT := _rTimeout, rTimer := _rTimer);
       // jump back
      _rStep := 10;

       
